# B&R Automation Studio project MotionTestBenchMaster (part 58)

```iecst
                               VAR_DOS_SEQ.Device.LSJ201.ALR := FALSE;                                                 (* STEP: 163 *)
                               VAR_DOS_SEQ.Device.LSJ201.WAIT_OFF := FALSE;
                               VAR_DOS_SEQ.Device.LSJ201.WAIT_ON := FALSE;

                               VAR_DOS_SEQ.Device.LSJ202.ALR := FALSE;                                                 (* STEP: 163 *)
                               VAR_DOS_SEQ.Device.LSJ202.WAIT_OFF := FALSE;
                               VAR_DOS_SEQ.Device.LSJ202.WAIT_ON := FALSE;

                               VAR_DOS_SEQ.Device.FSJ201.ALR := FALSE;                                                 (* STEP: 163 *)
                               VAR_DOS_SEQ.Device.FSJ201.WAIT_OFF := FALSE;
                               VAR_DOS_SEQ.Device.FSJ201.WAIT_ON := FALSE;

                               VAR_DOS_SEQ.Device.FSJ202.ALR := FALSE;                                                 (* STEP: 163 *)
                               VAR_DOS_SEQ.Device.FSJ202.WAIT_OFF := FALSE;
                               VAR_DOS_SEQ.Device.FSJ202.WAIT_ON := FALSE;

                               VAR_DOS_SEQ.Mem.PBAbortEnable := FALSE;                                                 (* STEP: 163 PB Abort Sequence Enable*)
                               VAR_DOS_SEQ.Mem.PBStopEnable := TRUE;                                                   (* STEP: 163 PB Stop Sequence Enable*)
                               VAR_DOS_SEQ.Mem.PBStartEnable := FALSE;                                                 (* STEP: 163 PB Start Sequence Enable*)
                               VAR_DOS_SEQ.Mem.ContainersStop := TRUE;                                                (* STEP: 163 *)
                               VAR_DOS_SEQ.Mem.MachineStart := FALSE;                                                  (* STEP: 163 *)
                               VAR_DOS_SEQ.Mem.MachineStop := FALSE;                                                   (* STEP: 163 *)
                               VAR_DOS_SEQ.Mem.DummyBottles := FALSE;                                                  (* STEP: 163 Dummy Bottle Install*)
                               VAR_DOS_SEQ.Mem.PositioningRequest := FALSE;                                            (* STEP: 163 Request of Cam Positioning at height SP of Sequncer*)
                               VAR_DOS_SEQ.Mem.COP_Cycle := FALSE;                                                     (* STEP: 163 COP Cycle Check Requested*)
                               VAR_DOS_SEQ.Mem.LapsCounter := FALSE;                                                   (* STEP: 163 *)
                               VAR_DOS_SEQ.Mem.ValveOpening := FALSE;                                                  (* STEP: 163 *)
                               VAR_DOS_SEQ.Mem.CopAfterCipRequest := FALSE;                                            (* STEP: 163 Request Of Cop After Cip*)

                               VAR_DOS_SEQ.ITC.CIP_CleaningRequest := FALSE;                                           (* STEP: 163 To CIP -> Request of Solution Sending*)
                               VAR_DOS_SEQ.ITC.CIP_Alarm := FALSE;                                                     (* STEP: 163 To CIP -> Critical Alarm Present*)
                               VAR_DOS_SEQ.ITC.CIP_RinseEnded := FALSE;                                                (* STEP: 163 To CIP -> Rinse Finished*)
                               VAR_DOS_SEQ.ITC.CIP_ChangeEnded := FALSE;                                               (* STEP: 163 To CIP -> Change Finished*)
                               VAR_DOS_SEQ.ITC.CIP_DrainRunning := FALSE;                                              (* STEP: 163 To CIP -> Drain Cycle Running*)
                               VAR_DOS_SEQ.ITC.CIP_RinseRunning := FALSE;                                              (* STEP: 163 To CIP -> Rinse Cycle Running*)
                               VAR_DOS_SEQ.ITC.CIP_CleaningRunning := FALSE;                                           (* STEP: 163 To CIP -> Cleaning Cycle Running*)
                               VAR_DOS_SEQ.ITC.CIP_DrainEnded := FALSE;                                                (* STEP: 163 To CIP -> Drain Finished*)
                               VAR_DOS_SEQ.ITC.CIP_FloodingEnded := FALSE;                                             (* STEP: 163 To CIP -> Flooding Finished*)
                               VAR_DOS_SEQ.ITC.CIP_FlipEnable := FALSE;                                                (* STEP: 163 *)
                               VAR_DOS_SEQ.ITC.CIP_CycleEnded := FALSE;                                                (* STEP: 163 *)

                               VAR_DOS_SEQ.ITC.PROD_ReadyForHeating := FALSE;                                          (* STEP: 163 To PASTO -> Filler Ready for Production (Heating)*)
                               VAR_DOS_SEQ.ITC.PROD_DoserInTemperature := FALSE;                                       (* STEP: 163 To PASTO -> Filler Temperature OK (After Heating)*)
                               VAR_DOS_SEQ.ITC.PROD_ProductRequest := FALSE;                                           (* STEP: 163 To PASTO -> Product Request*)
                               VAR_DOS_SEQ.ITC.PROD_DoserOnFillingMode := FALSE;                                       (* STEP: 163 To PASTO -> Product Consumend -Filling Valve Opening*)
                               VAR_DOS_SEQ.ITC.PROD_EndProductionCompleted := FALSE;                                   (* STEP: 163 To PASTO -> End Production Done*)
                               VAR_DOS_SEQ.ITC.PROD_ProductRecoveryEnd := FALSE;                                       (* STEP: 163 To PASTO -> Product Recovery End*)
                               VAR_DOS_SEQ.ITC.PROD_WaterRequestAfterProd := FALSE;                                    (* STEP: 163 To PASTO -> Water Request For Filler Rinse Afetr Production*)

                       164: (* MOTORIZATION - Operation Completed *)

                               VAR_DOS_SEQ.Device.PPJ201_PID.PID_Enable := FALSE;                                      (* STEP: 164 Doser Recovery Pump*)
                               VAR_DOS_SEQ.Device.PPJ201_PID.PID_Mode := FALSE;
                               VAR_DOS_SEQ.Device.PPJ201_PID.Auto_SP_Value := 0;
                               VAR_DOS_SEQ.Device.PPJ201_PID.FIX_Value := 0;

                               VAR_DOS_SEQ.Device.PPJ202_PID.PID_Enable := FALSE;                                      (* STEP: 164 Doser Recovery Pump*)
                               VAR_DOS_SEQ.Device.PPJ202_PID.PID_Mode := FALSE;
                               VAR_DOS_SEQ.Device.PPJ202_PID.Auto_SP_Value := 0;
                               VAR_DOS_SEQ.Device.PPJ202_PID.FIX_Value := 0;

                               VAR_DOS_SEQ.Device.PPJ203_PID.PID_Enable := FALSE;                                      (* STEP: 164 Diaphragm Pump for Recovery pulp*)
                               VAR_DOS_SEQ.Device.PPJ203_PID.PID_Mode := FALSE;
                               VAR_DOS_SEQ.Device.PPJ203_PID.Auto_SP_Value := 0;
                               VAR_DOS_SEQ.Device.PPJ203_PID.FIX_Value := 0;

                               VAR_DOS_SEQ.Device.MMJ201_PID.PID_Enable := FALSE;                                      (* STEP: 164 Shaker Motor*)
                               VAR_DOS_SEQ.Device.MMJ201_PID.PID_Mode := FALSE;
                               VAR_DOS_SEQ.Device.MMJ201_PID.Auto_SP_Value := 0;
                               VAR_DOS_SEQ.Device.MMJ201_PID.FIX_Value := 0;

                               VAR_DOS_SEQ.Device.RVJ201_PID.PID_Enable := FALSE;                                      (* STEP: 164 *)
                               VAR_DOS_SEQ.Device.RVJ201_PID.PID_Mode := FALSE;
                               VAR_DOS_SEQ.Device.RVJ201_PID.Auto_SP_Value := 0;
                               VAR_DOS_SEQ.Device.RVJ201_PID.FIX_Value := 0;

                               VAR_DOS_SEQ.Device.AVJ201.AutoCnd := FALSE;                                             (* STEP: 164 Inlet Valve*)
                               VAR_DOS_SEQ.Device.AVJ201.EnableCnd := FALSE;
                               VAR_DOS_SEQ.Device.AVJ210.AutoCnd := FALSE;                                             (* STEP: 164 Washing Duct Valve*)
                               VAR_DOS_SEQ.Device.AVJ210.EnableCnd := FALSE;
                               VAR_DOS_SEQ.Device.AVJ211.AutoCnd := FALSE;                                             (* STEP: 164 Sprayball Valve*)
                               VAR_DOS_SEQ.Device.AVJ211.EnableCnd := FALSE;
                               VAR_DOS_SEQ.Device.AVJ212.AutoCnd := FALSE;                                             (* STEP: 164 *)
                               VAR_DOS_SEQ.Device.AVJ212.EnableCnd := FALSE;
                               VAR_DOS_SEQ.Device.AVJ215.AutoCnd := FALSE;                                             (* STEP: 164 Atmospheric drain valve*)
                               VAR_DOS_SEQ.Device.AVJ215.EnableCnd := FALSE;
                               VAR_DOS_SEQ.Device.AVJ216.AutoCnd := FALSE;                                             (* STEP: 164 Recirculation Valve*)
                               VAR_DOS_SEQ.Device.AVJ216.EnableCnd := FALSE;
                               VAR_DOS_SEQ.Device.AVJ217.AutoCnd := FALSE;                                             (* STEP: 164 Tank Hema Drain Valve*)
                               VAR_DOS_SEQ.Device.AVJ217.EnableCnd := FALSE;
                               VAR_DOS_SEQ.Device.AVJ218.AutoCnd := FALSE;                                             (* STEP: 164 Recirculation Valve*)
                               VAR_DOS_SEQ.Device.AVJ218.EnableCnd := FALSE;
                               VAR_DOS_SEQ.Device.AVJ221.AutoCnd := FALSE;                                             (* STEP: 164 Inlet Loop Valve*)
                               VAR_DOS_SEQ.Device.AVJ221.EnableCnd := FALSE;
                               VAR_DOS_SEQ.Device.AVJ230.AutoCnd := FALSE;                                             (* STEP: 164 *)
                               VAR_DOS_SEQ.Device.AVJ230.EnableCnd := FALSE;
                               VAR_DOS_SEQ.Device.AVJ231.AutoCnd := FALSE;                                             (* STEP: 164 *)
                               VAR_DOS_SEQ.Device.AVJ231.EnableCnd := FALSE;
                               VAR_DOS_SEQ.Device.AVJ232.AutoCnd := FALSE;                                             (* STEP: 164 *)
                               VAR_DOS_SEQ.Device.AVJ232.EnableCnd := FALSE;
                               VAR_DOS_SEQ.Device.AVJ233.AutoCnd := FALSE;                                             (* STEP: 164 *)
                               VAR_DOS_SEQ.Device.AVJ233.EnableCnd := FALSE;
                               VAR_DOS_SEQ.Device.AVJ234.AutoCnd := FALSE;                                             (* STEP: 164 *)
                               VAR_DOS_SEQ.Device.AVJ234.EnableCnd := FALSE;
                               VAR_DOS_SEQ.Device.AVJ235.AutoCnd := FALSE;                                             (* STEP: 164 *)
                               VAR_DOS_SEQ.Device.AVJ235.EnableCnd := FALSE;

                               VAR_DOS_SEQ.Device.LTJ203.ALR_HighLimitEn := FALSE;                                     (* STEP: 164 Hema Tank Level*)
                               VAR_DOS_SEQ.Device.LTJ203.ALR_HighLimitSP := 0;
                               VAR_DOS_SEQ.Device.LTJ203.ALR_LowLimitEn := FALSE;
                               VAR_DOS_SEQ.Device.LTJ203.ALR_LowLimitSP := 0;
                               VAR_DOS_SEQ.Device.LTJ203.SP := 0;
                               VAR_DOS_SEQ.Device.LTJ203.CMP := 0;
                               VAR_DOS_SEQ.Device.LTJ203.MinDev := 0;
                               VAR_DOS_SEQ.Device.LTJ203.MaxDev := 0;

                               VAR_DOS_SEQ.Device.TTJ203.ALR_HighLimitEn := FALSE;                                     (* STEP: 164 Hema Tank Temperature*)
                               VAR_DOS_SEQ.Device.TTJ203.ALR_HighLimitSP := 0;
                               VAR_DOS_SEQ.Device.TTJ203.ALR_LowLimitEn := FALSE;
                               VAR_DOS_SEQ.Device.TTJ203.ALR_LowLimitSP := 0;
                               VAR_DOS_SEQ.Device.TTJ203.SP := 0;
                               VAR_DOS_SEQ.Device.TTJ203.CMP := 0;
                               VAR_DOS_SEQ.Device.TTJ203.MinDev := 0;
                               VAR_DOS_SEQ.Device.TTJ203.MaxDev := 0;

                               VAR_DOS_SEQ.Device.LSJ200.ALR := FALSE;                                                 (* STEP: 164 *)
                               VAR_DOS_SEQ.Device.LSJ200.WAIT_OFF := FALSE;
                               VAR_DOS_SEQ.Device.LSJ200.WAIT_ON := FALSE;

                               VAR_DOS_SEQ.Device.LSJ201.ALR := FALSE;                                                 (* STEP: 164 *)
                               VAR_DOS_SEQ.Device.LSJ201.WAIT_OFF := FALSE;
                               VAR_DOS_SEQ.Device.LSJ201.WAIT_ON := FALSE;

                               VAR_DOS_SEQ.Device.LSJ202.ALR := FALSE;                                                 (* STEP: 164 *)
                               VAR_DOS_SEQ.Device.LSJ202.WAIT_OFF := FALSE;
                               VAR_DOS_SEQ.Device.LSJ202.WAIT_ON := FALSE;

                               VAR_DOS_SEQ.Device.FSJ201.ALR := FALSE;                                                 (* STEP: 164 *)
                               VAR_DOS_SEQ.Device.FSJ201.WAIT_OFF := FALSE;
                               VAR_DOS_SEQ.Device.FSJ201.WAIT_ON := FALSE;

                               VAR_DOS_SEQ.Device.FSJ202.ALR := FALSE;                                                 (* STEP: 164 *)
                               VAR_DOS_SEQ.Device.FSJ202.WAIT_OFF := FALSE;
                               VAR_DOS_SEQ.Device.FSJ202.WAIT_ON := FALSE;

                               VAR_DOS_SEQ.Mem.PBAbortEnable := FALSE;                                                 (* STEP: 164 PB Abort Sequence Enable*)
                               VAR_DOS_SEQ.Mem.PBStopEnable := TRUE;                                                   (* STEP: 164 PB Stop Sequence Enable*)
                               VAR_DOS_SEQ.Mem.PBStartEnable := FALSE;                                                 (* STEP: 164 PB Start Sequence Enable*)
                               VAR_DOS_SEQ.Mem.ContainersStop := TRUE;                                                (* STEP: 164 *)
                               VAR_DOS_SEQ.Mem.MachineStart := FALSE;                                                  (* STEP: 164 *)
                               VAR_DOS_SEQ.Mem.MachineStop := FALSE;                                                   (* STEP: 164 *)
                               VAR_DOS_SEQ.Mem.DummyBottles := FALSE;                                                  (* STEP: 164 Dummy Bottle Install*)
                               VAR_DOS_SEQ.Mem.PositioningRequest := FALSE;                                            (* STEP: 164 Request of Cam Positioning at height SP of Sequncer*)
                               VAR_DOS_SEQ.Mem.COP_Cycle := FALSE;                                                     (* STEP: 164 COP Cycle Check Requested*)
                               VAR_DOS_SEQ.Mem.LapsCounter := FALSE;                                                   (* STEP: 164 *)
                               VAR_DOS_SEQ.Mem.ValveOpening := FALSE;                                                  (* STEP: 164 *)
                               VAR_DOS_SEQ.Mem.CopAfterCipRequest := FALSE;                                            (* STEP: 164 Request Of Cop After Cip*)

                               VAR_DOS_SEQ.ITC.CIP_CleaningRequest := FALSE;                                           (* STEP: 164 To CIP -> Request of Solution Sending*)
                               VAR_DOS_SEQ.ITC.CIP_Alarm := FALSE;                                                     (* STEP: 164 To CIP -> Critical Alarm Present*)
                               VAR_DOS_SEQ.ITC.CIP_RinseEnded := FALSE;                                                (* STEP: 164 To CIP -> Rinse Finished*)
                               VAR_DOS_SEQ.ITC.CIP_ChangeEnded := FALSE;                                               (* STEP: 164 To CIP -> Change Finished*)
                               VAR_DOS_SEQ.ITC.CIP_DrainRunning := FALSE;                                              (* STEP: 164 To CIP -> Drain Cycle Running*)
                               VAR_DOS_SEQ.ITC.CIP_RinseRunning := FALSE;                                              (* STEP: 164 To CIP -> Rinse Cycle Running*)
                               VAR_DOS_SEQ.ITC.CIP_CleaningRunning := FALSE;                                           (* STEP: 164 To CIP -> Cleaning Cycle Running*)
                               VAR_DOS_SEQ.ITC.CIP_DrainEnded := FALSE;                                                (* STEP: 164 To CIP -> Drain Finished*)
                               VAR_DOS_SEQ.ITC.CIP_FloodingEnded := FALSE;                                             (* STEP: 164 To CIP -> Flooding Finished*)
                               VAR_DOS_SEQ.ITC.CIP_FlipEnable := FALSE;                                                (* STEP: 164 *)
                               VAR_DOS_SEQ.ITC.CIP_CycleEnded := FALSE;                                                (* STEP: 164 *)

                               VAR_DOS_SEQ.ITC.PROD_ReadyForHeating := FALSE;                                          (* STEP: 164 To PASTO -> Filler Ready for Production (Heating)*)
                               VAR_DOS_SEQ.ITC.PROD_DoserInTemperature := FALSE;                                       (* STEP: 164 To PASTO -> Filler Temperature OK (After Heating)*)
                               VAR_DOS_SEQ.ITC.PROD_ProductRequest := FALSE;                                           (* STEP: 164 To PASTO -> Product Request*)
                               VAR_DOS_SEQ.ITC.PROD_DoserOnFillingMode := FALSE;                                       (* STEP: 164 To PASTO -> Product Consumend -Filling Valve Opening*)
                               VAR_DOS_SEQ.ITC.PROD_EndProductionCompleted := FALSE;                                   (* STEP: 164 To PASTO -> End Production Done*)
                               VAR_DOS_SEQ.ITC.PROD_ProductRecoveryEnd := FALSE;                                       (* STEP: 164 To PASTO -> Product Recovery End*)
                               VAR_DOS_SEQ.ITC.PROD_WaterRequestAfterProd := FALSE;                                    (* STEP: 164 To PASTO -> Water Request For Filler Rinse Afetr Production*)

                       165: (* MOTORIZATION - Error *)

                               VAR_DOS_SEQ.Device.PPJ201_PID.PID_Enable := FALSE;                                      (* STEP: 165 Doser Recovery Pump*)
                               VAR_DOS_SEQ.Device.PPJ201_PID.PID_Mode := FALSE;
                               VAR_DOS_SEQ.Device.PPJ201_PID.Auto_SP_Value := 0;
                               VAR_DOS_SEQ.Device.PPJ201_PID.FIX_Value := 0;

                               VAR_DOS_SEQ.Device.PPJ202_PID.PID_Enable := FALSE;                                      (* STEP: 165 Doser Recovery Pump*)
                               VAR_DOS_SEQ.Device.PPJ202_PID.PID_Mode := FALSE;
                               VAR_DOS_SEQ.Device.PPJ202_PID.Auto_SP_Value := 0;
                               VAR_DOS_SEQ.Device.PPJ202_PID.FIX_Value := 0;

                               VAR_DOS_SEQ.Device.PPJ203_PID.PID_Enable := FALSE;                                      (* STEP: 165 Diaphragm Pump for Recovery pulp*)
                               VAR_DOS_SEQ.Device.PPJ203_PID.PID_Mode := FALSE;
                               VAR_DOS_SEQ.Device.PPJ203_PID.Auto_SP_Value := 0;
                               VAR_DOS_SEQ.Device.PPJ203_PID.FIX_Value := 0;

                               VAR_DOS_SEQ.Device.MMJ201_PID.PID_Enable := FALSE;                                      (* STEP: 165 Shaker Motor*)
                               VAR_DOS_SEQ.Device.MMJ201_PID.PID_Mode := FALSE;
                               VAR_DOS_SEQ.Device.MMJ201_PID.Auto_SP_Value := 0;
                               VAR_DOS_SEQ.Device.MMJ201_PID.FIX_Value := 0;

                               VAR_DOS_SEQ.Device.RVJ201_PID.PID_Enable := FALSE;                                      (* STEP: 165 *)
                               VAR_DOS_SEQ.Device.RVJ201_PID.PID_Mode := FALSE;
                               VAR_DOS_SEQ.Device.RVJ201_PID.Auto_SP_Value := 0;
                               VAR_DOS_SEQ.Device.RVJ201_PID.FIX_Value := 0;

                               VAR_DOS_SEQ.Device.AVJ201.AutoCnd := FALSE;                                             (* STEP: 165 Inlet Valve*)
                               VAR_DOS_SEQ.Device.AVJ201.EnableCnd := FALSE;
                               VAR_DOS_SEQ.Device.AVJ210.AutoCnd := FALSE;                                             (* STEP: 165 Washing Duct Valve*)
                               VAR_DOS_SEQ.Device.AVJ210.EnableCnd := FALSE;
                               VAR_DOS_SEQ.Device.AVJ211.AutoCnd := FALSE;                                             (* STEP: 165 Sprayball Valve*)
                               VAR_DOS_SEQ.Device.AVJ211.EnableCnd := FALSE;
                               VAR_DOS_SEQ.Device.AVJ212.AutoCnd := FALSE;                                             (* STEP: 165 *)
                               VAR_DOS_SEQ.Device.AVJ212.EnableCnd := FALSE;
                               VAR_DOS_SEQ.Device.AVJ215.AutoCnd := FALSE;                                             (* STEP: 165 Atmospheric drain valve*)
                               VAR_DOS_SEQ.Device.AVJ215.EnableCnd := FALSE;
                               VAR_DOS_SEQ.Device.AVJ216.AutoCnd := FALSE;                                             (* STEP: 165 Recirculation Valve*)
                               VAR_DOS_SEQ.Device.AVJ216.EnableCnd := FALSE;
                               VAR_DOS_SEQ.Device.AVJ217.AutoCnd := FALSE;                                             (* STEP: 165 Tank Hema Drain Valve*)
                               VAR_DOS_SEQ.Device.AVJ217.EnableCnd := FALSE;
                               VAR_DOS_SEQ.Device.AVJ218.AutoCnd := FALSE;                                             (* STEP: 165 Recirculation Valve*)
                               VAR_DOS_SEQ.Device.AVJ218.EnableCnd := FALSE;
                               VAR_DOS_SEQ.Device.AVJ221.AutoCnd := FALSE;                                             (* STEP: 165 Inlet Loop Valve*)
                               VAR_DOS_SEQ.Device.AVJ221.EnableCnd := FALSE;
                               VAR_DOS_SEQ.Device.AVJ230.AutoCnd := FALSE;                                             (* STEP: 165 *)
                               VAR_DOS_SEQ.Device.AVJ230.EnableCnd := FALSE;
                               VAR_DOS_SEQ.Device.AVJ231.AutoCnd := FALSE;                                             (* STEP: 165 *)
                               VAR_DOS_SEQ.Device.AVJ231.EnableCnd := FALSE;
                               VAR_DOS_SEQ.Device.AVJ232.AutoCnd := FALSE;                                             (* STEP: 165 *)
                               VAR_DOS_SEQ.Device.AVJ232.EnableCnd := FALSE;
                               VAR_DOS_SEQ.Device.AVJ233.AutoCnd := FALSE;                                             (* STEP: 165 *)
                               VAR_DOS_SEQ.Device.AVJ233.EnableCnd := FALSE;
                               VAR_DOS_SEQ.Device.AVJ234.AutoCnd := FALSE;                                             (* STEP: 165 *)
                               VAR_DOS_SEQ.Device.AVJ234.EnableCnd := FALSE;
                               VAR_DOS_SEQ.Device.AVJ235.AutoCnd := FALSE;                                             (* STEP: 165 *)
                               VAR_DOS_SEQ.Device.AVJ235.EnableCnd := FALSE;

                               VAR_DOS_SEQ.Device.LTJ203.ALR_HighLimitEn := FALSE;                                     (* STEP: 165 Hema Tank Level*)
                               VAR_DOS_SEQ.Device.LTJ203.ALR_HighLimitSP := 0;
                               VAR_DOS_SEQ.Device.LTJ203.ALR_LowLimitEn := FALSE;
                               VAR_DOS_SEQ.Device.LTJ203.ALR_LowLimitSP := 0;
                               VAR_DOS_SEQ.Device.LTJ203.SP := 0;
                               VAR_DOS_SEQ.Device.LTJ203.CMP := 0;
                               VAR_DOS_SEQ.Device.LTJ203.MinDev := 0;
                               VAR_DOS_SEQ.Device.LTJ203.MaxDev := 0;

                               VAR_DOS_SEQ.Device.TTJ203.ALR_HighLimitEn := FALSE;                                     (* STEP: 165 Hema Tank Temperature*)
                               VAR_DOS_SEQ.Device.TTJ203.ALR_HighLimitSP := 0;
                               VAR_DOS_SEQ.Device.TTJ203.ALR_LowLimitEn := FALSE;
                               VAR_DOS_SEQ.Device.TTJ203.ALR_LowLimitSP := 0;
                               VAR_DOS_SEQ.Device.TTJ203.SP := 0;
                               VAR_DOS_SEQ.Device.TTJ203.CMP := 0;
                               VAR_DOS_SEQ.Device.TTJ203.MinDev := 0;
                               VAR_DOS_SEQ.Device.TTJ203.MaxDev := 0;

                               VAR_DOS_SEQ.Device.LSJ200.ALR := FALSE;                                                 (* STEP: 165 *)
                               VAR_DOS_SEQ.Device.LSJ200.WAIT_OFF := FALSE;
                               VAR_DOS_SEQ.Device.LSJ200.WAIT_ON := FALSE;

                               VAR_DOS_SEQ.Device.LSJ201.ALR := FALSE;                                                 (* STEP: 165 *)
                               VAR_DOS_SEQ.Device.LSJ201.WAIT_OFF := FALSE;
                               VAR_DOS_SEQ.Device.LSJ201.WAIT_ON := FALSE;

                               VAR_DOS_SEQ.Device.LSJ202.ALR := FALSE;                                                 (* STEP: 165 *)
                               VAR_DOS_SEQ.Device.LSJ202.WAIT_OFF := FALSE;
                               VAR_DOS_SEQ.Device.LSJ202.WAIT_ON := FALSE;

                               VAR_DOS_SEQ.Device.FSJ201.ALR := FALSE;                                                 (* STEP: 165 *)
                               VAR_DOS_SEQ.Device.FSJ201.WAIT_OFF := FALSE;
                               VAR_DOS_SEQ.Device.FSJ201.WAIT_ON := FALSE;

                               VAR_DOS_SEQ.Device.FSJ202.ALR := FALSE;                                                 (* STEP: 165 *)
                               VAR_DOS_SEQ.Device.FSJ202.WAIT_OFF := FALSE;
                               VAR_DOS_SEQ.Device.FSJ202.WAIT_ON := FALSE;

                               VAR_DOS_SEQ.Mem.PBAbortEnable := TRUE;                                                 (* STEP: 165 PB Abort Sequence Enable*)
                               VAR_DOS_SEQ.Mem.PBStopEnable := TRUE;                                                   (* STEP: 165 PB Stop Sequence Enable*)
                               VAR_DOS_SEQ.Mem.PBStartEnable := FALSE;                                                 (* STEP: 165 PB Start Sequence Enable*)
                               VAR_DOS_SEQ.Mem.ContainersStop := TRUE;                                                (* STEP: 165 *)
                               VAR_DOS_SEQ.Mem.MachineStart := FALSE;                                                  (* STEP: 165 *)
                               VAR_DOS_SEQ.Mem.MachineStop := FALSE;                                                   (* STEP: 165 *)
                               VAR_DOS_SEQ.Mem.DummyBottles := FALSE;                                                  (* STEP: 165 Dummy Bottle Install*)
                               VAR_DOS_SEQ.Mem.PositioningRequest := FALSE;                                            (* STEP: 165 Request of Cam Positioning at height SP of Sequncer*)
                               VAR_DOS_SEQ.Mem.COP_Cycle := FALSE;                                                     (* STEP: 165 COP Cycle Check Requested*)
                               VAR_DOS_SEQ.Mem.LapsCounter := FALSE;                                                   (* STEP: 165 *)
                               VAR_DOS_SEQ.Mem.ValveOpening := FALSE;                                                  (* STEP: 165 *)
                               VAR_DOS_SEQ.Mem.CopAfterCipRequest := FALSE;                                            (* STEP: 165 Request Of Cop After Cip*)

                               VAR_DOS_SEQ.ITC.CIP_CleaningRequest := FALSE;                                           (* STEP: 165 To CIP -> Request of Solution Sending*)
                               VAR_DOS_SEQ.ITC.CIP_Alarm := FALSE;                                                     (* STEP: 165 To CIP -> Critical Alarm Present*)
                               VAR_DOS_SEQ.ITC.CIP_RinseEnded := FALSE;                                                (* STEP: 165 To CIP -> Rinse Finished*)
                               VAR_DOS_SEQ.ITC.CIP_ChangeEnded := FALSE;                                               (* STEP: 165 To CIP -> Change Finished*)
                               VAR_DOS_SEQ.ITC.CIP_DrainRunning := FALSE;                                              (* STEP: 165 To CIP -> Drain Cycle Running*)
                               VAR_DOS_SEQ.ITC.CIP_RinseRunning := FALSE;                                              (* STEP: 165 To CIP -> Rinse Cycle Running*)
                               VAR_DOS_SEQ.ITC.CIP_CleaningRunning := FALSE;                                           (* STEP: 165 To CIP -> Cleaning Cycle Running*)
                               VAR_DOS_SEQ.ITC.CIP_DrainEnded := FALSE;                                                (* STEP: 165 To CIP -> Drain Finished*)
                               VAR_DOS_SEQ.ITC.CIP_FloodingEnded := FALSE;                                             (* STEP: 165 To CIP -> Flooding Finished*)
                               VAR_DOS_SEQ.ITC.CIP_FlipEnable := FALSE;                                                (* STEP: 165 *)
                               VAR_DOS_SEQ.ITC.CIP_CycleEnded := FALSE;                                                (* STEP: 165 *)

                               VAR_DOS_SEQ.ITC.PROD_ReadyForHeating := FALSE;                                          (* STEP: 165 To PASTO -> Filler Ready for Production (Heating)*)
                               VAR_DOS_SEQ.ITC.PROD_DoserInTemperature := FALSE;                                       (* STEP: 165 To PASTO -> Filler Temperature OK (After Heating)*)
                               VAR_DOS_SEQ.ITC.PROD_ProductRequest := FALSE;                                           (* STEP: 165 To PASTO -> Product Request*)
                               VAR_DOS_SEQ.ITC.PROD_DoserOnFillingMode := FALSE;                                       (* STEP: 165 To PASTO -> Product Consumend -Filling Valve Opening*)
                               VAR_DOS_SEQ.ITC.PROD_EndProductionCompleted := FALSE;                                   (* STEP: 165 To PASTO -> End Production Done*)
                               VAR_DOS_SEQ.ITC.PROD_ProductRecoveryEnd := FALSE;                                       (* STEP: 165 To PASTO -> Product Recovery End*)
                               VAR_DOS_SEQ.ITC.PROD_WaterRequestAfterProd := FALSE;                                    (* STEP: 165 To PASTO -> Water Request For Filler Rinse Afetr Production*)

                       166..169: (* Spare Steps *)

                       170: (* PRODUCTION - Doser Excluded *)

                               VAR_DOS_SEQ.Device.PPJ201_PID.PID_Enable := FALSE;                                      (* STEP: 170 Doser Recovery Pump*)
                               VAR_DOS_SEQ.Device.PPJ201_PID.PID_Mode := FALSE;
                               VAR_DOS_SEQ.Device.PPJ201_PID.Auto_SP_Value := 0;
                               VAR_DOS_SEQ.Device.PPJ201_PID.FIX_Value := 0;

                               VAR_DOS_SEQ.Device.PPJ202_PID.PID_Enable := FALSE;                                      (* STEP: 170 Doser Recovery Pump*)
                               VAR_DOS_SEQ.Device.PPJ202_PID.PID_Mode := FALSE;
                               VAR_DOS_SEQ.Device.PPJ202_PID.Auto_SP_Value := 0;
                               VAR_DOS_SEQ.Device.PPJ202_PID.FIX_Value := 0;

                               VAR_DOS_SEQ.Device.PPJ203_PID.PID_Enable := FALSE;                                      (* STEP: 170 Diaphragm Pump for Recovery pulp*)
                               VAR_DOS_SEQ.Device.PPJ203_PID.PID_Mode := FALSE;
                               VAR_DOS_SEQ.Device.PPJ203_PID.Auto_SP_Value := 0;
                               VAR_DOS_SEQ.Device.PPJ203_PID.FIX_Value := 0;

                               VAR_DOS_SEQ.Device.MMJ201_PID.PID_Enable := FALSE;                                      (* STEP: 170 Shaker Motor*)
                               VAR_DOS_SEQ.Device.MMJ201_PID.PID_Mode := FALSE;
                               VAR_DOS_SEQ.Device.MMJ201_PID.Auto_SP_Value := 0;
                               VAR_DOS_SEQ.Device.MMJ201_PID.FIX_Value := 0;

                               VAR_DOS_SEQ.Device.RVJ201_PID.PID_Enable := FALSE;                                      (* STEP: 170 *)
                               VAR_DOS_SEQ.Device.RVJ201_PID.PID_Mode := FALSE;
                               VAR_DOS_SEQ.Device.RVJ201_PID.Auto_SP_Value := 0;
                               VAR_DOS_SEQ.Device.RVJ201_PID.FIX_Value := 0;

                               VAR_DOS_SEQ.Device.AVJ201.AutoCnd := FALSE;                                             (* STEP: 170 Inlet Valve*)
                               VAR_DOS_SEQ.Device.AVJ201.EnableCnd := FALSE;
                               VAR_DOS_SEQ.Device.AVJ210.AutoCnd := FALSE;                                             (* STEP: 170 Washing Duct Valve*)
                               VAR_DOS_SEQ.Device.AVJ210.EnableCnd := FALSE;
                               VAR_DOS_SEQ.Device.AVJ211.AutoCnd := FALSE;                                             (* STEP: 170 Sprayball Valve*)
                               VAR_DOS_SEQ.Device.AVJ211.EnableCnd := FALSE;
                               VAR_DOS_SEQ.Device.AVJ212.AutoCnd := FALSE;                                             (* STEP: 170 *)
                               VAR_DOS_SEQ.Device.AVJ212.EnableCnd := FALSE;
                               VAR_DOS_SEQ.Device.AVJ215.AutoCnd := FALSE;                                             (* STEP: 170 Atmospheric drain valve*)
                               VAR_DOS_SEQ.Device.AVJ215.EnableCnd := FALSE;
                               VAR_DOS_SEQ.Device.AVJ216.AutoCnd := FALSE;                                             (* STEP: 170 Recirculation Valve*)
                               VAR_DOS_SEQ.Device.AVJ216.EnableCnd := FALSE;
                               VAR_DOS_SEQ.Device.AVJ217.AutoCnd := FALSE;                                             (* STEP: 170 Tank Hema Drain Valve*)
                               VAR_DOS_SEQ.Device.AVJ217.EnableCnd := FALSE;
                               VAR_DOS_SEQ.Device.AVJ218.AutoCnd := FALSE;                                             (* STEP: 170 Recirculation Valve*)
                               VAR_DOS_SEQ.Device.AVJ218.EnableCnd := FALSE;
                               VAR_DOS_SEQ.Device.AVJ221.AutoCnd := FALSE;                                             (* STEP: 170 Inlet Loop Valve*)
                               VAR_DOS_SEQ.Device.AVJ221.EnableCnd := FALSE;
                               VAR_DOS_SEQ.Device.AVJ230.AutoCnd := FALSE;                                             (* STEP: 170 *)
                               VAR_DOS_SEQ.Device.AVJ230.EnableCnd := FALSE;
                               VAR_DOS_SEQ.Device.AVJ231.AutoCnd := FALSE;                                             (* STEP: 170 *)
                               VAR_DOS_SEQ.Device.AVJ231.EnableCnd := FALSE;
                               VAR_DOS_SEQ.Device.AVJ232.AutoCnd := FALSE;                                             (* STEP: 170 *)
                               VAR_DOS_SEQ.Device.AVJ232.EnableCnd := FALSE;
                               VAR_DOS_SEQ.Device.AVJ233.AutoCnd := FALSE;                                             (* STEP: 170 *)
                               VAR_DOS_SEQ.Device.AVJ233.EnableCnd := FALSE;
                               VAR_DOS_SEQ.Device.AVJ234.AutoCnd := FALSE;                                             (* STEP: 170 *)
                               VAR_DOS_SEQ.Device.AVJ234.EnableCnd := FALSE;
                               VAR_DOS_SEQ.Device.AVJ235.AutoCnd := FALSE;                                             (* STEP: 170 *)
                               VAR_DOS_SEQ.Device.AVJ235.EnableCnd := FALSE;

                               VAR_DOS_SEQ.Device.LTJ203.ALR_HighLimitEn := FALSE;                                     (* STEP: 170 Hema Tank Level*)
                               VAR_DOS_SEQ.Device.LTJ203.ALR_HighLimitSP := 0;
                               VAR_DOS_SEQ.Device.LTJ203.ALR_LowLimitEn := FALSE;
                               VAR_DOS_SEQ.Device.LTJ203.ALR_LowLimitSP := 0;
                               VAR_DOS_SEQ.Device.LTJ203.SP := 0;
                               VAR_DOS_SEQ.Device.LTJ203.CMP := 0;
                               VAR_DOS_SEQ.Device.LTJ203.MinDev := 0;
                               VAR_DOS_SEQ.Device.LTJ203.MaxDev := 0;

                               VAR_DOS_SEQ.Device.TTJ203.ALR_HighLimitEn := FALSE;                                     (* STEP: 170 Hema Tank Temperature*)
                               VAR_DOS_SEQ.Device.TTJ203.ALR_HighLimitSP := 0;
                               VAR_DOS_SEQ.Device.TTJ203.ALR_LowLimitEn := FALSE;
                               VAR_DOS_SEQ.Device.TTJ203.ALR_LowLimitSP := 0;
                               VAR_DOS_SEQ.Device.TTJ203.SP := 0;
                               VAR_DOS_SEQ.Device.TTJ203.CMP := 0;
                               VAR_DOS_SEQ.Device.TTJ203.MinDev := 0;
                               VAR_DOS_SEQ.Device.TTJ203.MaxDev := 0;

                               VAR_DOS_SEQ.Device.LSJ200.ALR := FALSE;                                                 (* STEP: 170 *)
                               VAR_DOS_SEQ.Device.LSJ200.WAIT_OFF := FALSE;
                               VAR_DOS_SEQ.Device.LSJ200.WAIT_ON := FALSE;

                               VAR_DOS_SEQ.Device.LSJ201.ALR := FALSE;                                                 (* STEP: 170 *)
                               VAR_DOS_SEQ.Device.LSJ201.WAIT_OFF := FALSE;
                               VAR_DOS_SEQ.Device.LSJ201.WAIT_ON := FALSE;

                               VAR_DOS_SEQ.Device.LSJ202.ALR := FALSE;                                                 (* STEP: 170 *)
                               VAR_DOS_SEQ.Device.LSJ202.WAIT_OFF := FALSE;
                               VAR_DOS_SEQ.Device.LSJ202.WAIT_ON := FALSE;

                               VAR_DOS_SEQ.Device.FSJ201.ALR := FALSE;                                                 (* STEP: 170 *)
                               VAR_DOS_SEQ.Device.FSJ201.WAIT_OFF := FALSE;
                               VAR_DOS_SEQ.Device.FSJ201.WAIT_ON := FALSE;

                               VAR_DOS_SEQ.Device.FSJ202.ALR := FALSE;                                                 (* STEP: 170 *)
                               VAR_DOS_SEQ.Device.FSJ202.WAIT_OFF := FALSE;
                               VAR_DOS_SEQ.Device.FSJ202.WAIT_ON := FALSE;

                               VAR_DOS_SEQ.Mem.PBAbortEnable := FALSE;                                                 (* STEP: 170 PB Abort Sequence Enable*)
                               VAR_DOS_SEQ.Mem.PBStopEnable := FALSE;                                                   (* STEP: 170 PB Stop Sequence Enable*)
                               VAR_DOS_SEQ.Mem.PBStartEnable := FALSE;                                                 (* STEP: 170 PB Start Sequence Enable*)
                               VAR_DOS_SEQ.Mem.ContainersStop := FALSE;                                                (* STEP: 170 *)
                               VAR_DOS_SEQ.Mem.MachineStart := FALSE;                                                  (* STEP: 170 *)
                               VAR_DOS_SEQ.Mem.MachineStop := FALSE;                                                   (* STEP: 170 *)
                               VAR_DOS_SEQ.Mem.DummyBottles := FALSE;                                                  (* STEP: 170 Dummy Bottle Install*)
                               VAR_DOS_SEQ.Mem.PositioningRequest := FALSE;                                            (* STEP: 170 Request of Cam Positioning at height SP of Sequncer*)
                               VAR_DOS_SEQ.Mem.COP_Cycle := FALSE;                                                     (* STEP: 170 COP Cycle Check Requested*)
                               VAR_DOS_SEQ.Mem.LapsCounter := FALSE;                                                   (* STEP: 170 *)
                               VAR_DOS_SEQ.Mem.ValveOpening := FALSE;                                                  (* STEP: 170 *)
                               VAR_DOS_SEQ.Mem.CopAfterCipRequest := FALSE;                                            (* STEP: 170 Request Of Cop After Cip*)

                               VAR_DOS_SEQ.ITC.CIP_CleaningRequest := FALSE;                                           (* STEP: 170 To CIP -> Request of Solution Sending*)
                               VAR_DOS_SEQ.ITC.CIP_Alarm := FALSE;                                                     (* STEP: 170 To CIP -> Critical Alarm Present*)
                               VAR_DOS_SEQ.ITC.CIP_RinseEnded := FALSE;                                                (* STEP: 170 To CIP -> Rinse Finished*)
                               VAR_DOS_SEQ.ITC.CIP_ChangeEnded := FALSE;                                               (* STEP: 170 To CIP -> Change Finished*)
                               VAR_DOS_SEQ.ITC.CIP_DrainRunning := FALSE;                                              (* STEP: 170 To CIP -> Drain Cycle Running*)
                               VAR_DOS_SEQ.ITC.CIP_RinseRunning := FALSE;                                              (* STEP: 170 To CIP -> Rinse Cycle Running*)
                               VAR_DOS_SEQ.ITC.CIP_CleaningRunning := FALSE;                                           (* STEP: 170 To CIP -> Cleaning Cycle Running*)
                               VAR_DOS_SEQ.ITC.CIP_DrainEnded := FALSE;                                                (* STEP: 170 To CIP -> Drain Finished*)
                               VAR_DOS_SEQ.ITC.CIP_FloodingEnded := FALSE;                                             (* STEP: 170 To CIP -> Flooding Finished*)
                               VAR_DOS_SEQ.ITC.CIP_FlipEnable := FALSE;                                                (* STEP: 170 *)
                               VAR_DOS_SEQ.ITC.CIP_CycleEnded := FALSE;                                                (* STEP: 170 *)

                               VAR_DOS_SEQ.ITC.PROD_ReadyForHeating := FALSE;                                          (* STEP: 170 To PASTO -> Filler Ready for Production (Heating)*)
                               VAR_DOS_SEQ.ITC.PROD_DoserInTemperature := FALSE;                                       (* STEP: 170 To PASTO -> Filler Temperature OK (After Heating)*)
                               VAR_DOS_SEQ.ITC.PROD_ProductRequest := FALSE;                                           (* STEP: 170 To PASTO -> Product Request*)
                               VAR_DOS_SEQ.ITC.PROD_DoserOnFillingMode := FALSE;                                       (* STEP: 170 To PASTO -> Product Consumend -Filling Valve Opening*)
                               VAR_DOS_SEQ.ITC.PROD_EndProductionCompleted := FALSE;                                   (* STEP: 170 To PASTO -> End Production Done*)
                               VAR_DOS_SEQ.ITC.PROD_ProductRecoveryEnd := FALSE;                                       (* STEP: 170 To PASTO -> Product Recovery End*)
                               VAR_DOS_SEQ.ITC.PROD_WaterRequestAfterProd := FALSE;                                    (* STEP: 170 To PASTO -> Water Request For Filler Rinse Afetr Production*)

                       171..200: (* Spare Steps *)

               END_CASE
END_ACTION
```

#### DOS_StepStatus.st
```iecst
ACTION DOS_StepStatus:
	//MODE
	VAR_DOS_ModeWait					:= VAR_DOS_SeqPermanent.SeqActualStep = 0;
	VAR_DOS_ModeProduction				:= VAR_DOS_SeqPermanent.SeqMode1.0;
	VAR_DOS_ModeCip						:= VAR_DOS_SeqPermanent.SeqMode1.1;
	VAR_DOS_ModeRinse					:= VAR_DOS_SeqPermanent.SeqMode1.2;
	VAR_DOS_ModeDrain					:= VAR_DOS_SeqPermanent.SeqMode1.3;
	VAR_DOS_ModeCop						:= VAR_DOS_SeqPermanent.SeqMode1.4;
	VAR_DOS_ModePositioning				:= VAR_DOS_SeqPermanent.SeqMode1.5;
	VAR_DOS_ModeBypass					:= VAR_DOS_SeqPermanent.SeqMode1.6;
	VAR_DOS_ModePositionRequest			:= VAR_DOS_SeqPermanent.SeqMode1.7;
	VAR_DOS_ModeProductionExcluded		:= VAR_DOS_SeqPermanent.SeqMode1.8;
	VAR_DOS_MemProdDrain				:= VAR_DOS_SeqPermanent.SeqMode2.0;
	VAR_DOS_ModeWaitOperator			:= FALSE;

	VAR_DOS_MemDoserByPassed			:= VAR_DOS_SeqPermanent.SeqMode2.2;
	VAR_DOS_MemDoserIncluded			:= VAR_DOS_SeqPermanent.SeqMode2.3;

	VAR_DOS_MemDoserAxisOn				:= VAR_DOS_SeqPermanent.SeqMode2.4;
	VAR_DOS_MemDoserAxisOff				:= VAR_DOS_SeqPermanent.SeqMode2.5;
	VAR_DOS_MemFillerAxisOffReq			:= VAR_DOS_SeqPermanent.SeqMode2.6;

	//STEP PRODUCTION
	VAR_DOS_StepProdHeating				:= VAR_DOS_SEQ_Step.StepActual > 6 AND VAR_DOS_SeqActualStep < 15;
	VAR_DOS_StepProdProducing			:= VAR_DOS_SEQ_Step.StepActual = 35 OR VAR_DOS_SEQ_Step.StepActual = 37 OR VAR_DOS_SEQ_Step.StepActual = 38 OR
											VAR_DOS_SEQ_Step.StepActual = 22 OR VAR_DOS_SEQ_Step.StepActual = 23 OR VAR_DOS_SEQ_Step.StepActual = 30;
	VAR_DOS_StepProdLowLevel			:= VAR_DOS_SEQ_Step.StepActual = 37;
	VAR_DOS_StepProdRecovery			:= VAR_DOS_SEQ_Step.StepActual = 40;
	VAR_DOS_StepProdStopped				:= VAR_DOS_SEQ_Step.StepActual = 55;
	VAR_DOS_StepProdEndProduction		:= VAR_DOS_SEQ_Step.StepActual >= 46 AND VAR_DOS_SeqActualStep <= 52;
	VAR_DOS_StepProdAborted				:= VAR_DOS_SEQ_Step.StepActual = 0;

	//STEP CIP
	VAR_DOS_StepCipCleaning				:= VAR_DOS_SEQ_Step.StepActual > 73 AND VAR_DOS_SeqActualStep <=79;		//<	83
	VAR_DOS_StepCipDraining				:= VAR_DOS_SEQ_Step.StepActual >= 86 AND VAR_DOS_SeqActualStep <= 87;
	VAR_DOS_StepCipRecovery				:= VAR_DOS_SEQ_Step.StepActual = 82;
	VAR_DOS_StepCipStopped				:= VAR_DOS_SEQ_Step.StepActual = 95;
	VAR_DOS_StepCipAborted				:= VAR_DOS_SEQ_Step.StepActual = 96 OR VAR_DOS_SEQ_Step.StepActual = 0;
	VAR_DOS_StepCipEnded				:= VAR_DOS_SEQ_Step.StepActual = 88;
	VAR_DOS_StepCipFillerStartEnable	:= VAR_DOS_SEQ_Step.StepActual = 60 OR VAR_DOS_SeqActualStep = 61; //Segnale per SKID

	//STEP RINSE
	VAR_DOS_StepRinseReq				:=  VAR_DOS_SEQ_Step.StepActual >= 101 AND VAR_DOS_SeqActualStep <=106;
	VAR_DOS_StepRinseInExecution		:=  VAR_DOS_SEQ_Step.StepActual >= 101 AND VAR_DOS_SeqActualStep <=109;
	VAR_DOS_StepRinseAborted			:= VAR_DOS_SEQ_Step.StepActual = 0;
	VAR_DOS_StepRinseStopped			:= VAR_DOS_SEQ_Step.StepActual = 115;

	//STEP DRAIN
	VAR_DOS_StepDrainStopped			:= VAR_DOS_SEQ_Step.StepActual = 135;
	VAR_DOS_StepDrainAborted			:= VAR_DOS_SEQ_Step.StepActual = 0;

	//STEP COP
	VAR_DOS_StepCopRunning				:= VAR_DOS_SEQ_Step.StepActual = 90;

	//STEP BYPASS
	VAR_DOS_StepCamPositioning				:= VAR_DOS_SeqActualStep >= 150 AND VAR_DOS_SeqActualStep <= 155;
	VAR_DOS_StepCamPosRequest				:= VAR_DOS_SeqActualStep = 151;
	VAR_DOS_StepCamPosInProgress			:= VAR_DOS_SeqActualStep >= 151 AND VAR_DOS_SeqActualStep <= 154;
	VAR_DOS_StepBypassAborted				:= VAR_DOS_SeqActualStep = 0;

	//STEP MOTION
	VAR_DOS_StepMotorization				:= VAR_DOS_SeqActualStep >= 161 AND VAR_DOS_SeqActualStep <= 163;
END_ACTION
```

#### DOS_ValvesLogic.st
```iecst
ACTION DOS_ValvesLogic:

	VAR_DOS_ValveEnable := OPS.DataOut.EmergencyOk AND OPS.DataOut.GeneralAirOn AND OPS.DataOut.DoorsOk;

//AVJ201
	AVJ[201].IN_Enable		:= VAR_DOS_ValveEnable;
	AVJ[201].IN_AutoCnd		:= VAR_DOS_SEQ.Device.AVJ201.AutoCnd;
	AVJ[201].IN_EnableCnd	:= VAR_DOS_SEQ.Device.AVJ201.EnableCnd;
	AVJ[201].IN_Cnd 		:= (NOT LTJ[203].OUT_SpReached AND PstFlr.ProductAvailable AND VAR_DOS_StepProdProducing) OR
	                           (NOT LTJ[203].OUT_SpReached AND PstFlr.HeatingWithWater AND VAR_DOS_StepProdHeating) OR
                               (NOT LTJ[203].OUT_SpReached AND VAR_DOS_StepCipCleaning) OR
								(NOT LTJ[203].OUT_SpReached AND VAR_DOS_StepRinseReq) OR
								(NOT LTJ[203].OUT_SpReached AND VAR_DOS_SEQ_Step.StepActual = 46 AND  PstFlr.ProductAvailable); //46
	AVJ[201].IN_ManEn		:= TRUE;
	AVJ[201].IN_MaskEn		:= TRUE;

//AVJ210
	AVJ[210].IN_Enable		:= VAR_DOS_ValveEnable;
	AVJ[210].IN_AutoCnd		:= VAR_DOS_SEQ.Device.AVJ210.AutoCnd;
	AVJ[210].IN_EnableCnd	:= VAR_DOS_SEQ.Device.AVJ210.EnableCnd;
	AVJ[210].IN_Cnd 		:= FALSE;
	AVJ[210].IN_ManEn		:= TRUE;
	AVJ[210].IN_MaskEn		:= TRUE;

//AVJ211
	AVJ[211].IN_Enable		:= VAR_DOS_ValveEnable;
	AVJ[211].IN_AutoCnd		:= VAR_DOS_SEQ.Device.AVJ211.AutoCnd;
	AVJ[211].IN_EnableCnd	:= VAR_DOS_SEQ.Device.AVJ211.EnableCnd;
	AVJ[211].IN_Cnd 		:= NOT LTJ[203].OUT_HighLimit;
	AVJ[211].IN_ManEn		:= TRUE;
	AVJ[211].IN_MaskEn		:= TRUE;

//AVJ212
	AVJ[212].IN_Enable		:= VAR_DOS_ValveEnable;
	AVJ[212].IN_AutoCnd		:= VAR_DOS_SEQ.Device.AVJ212.AutoCnd;
	AVJ[212].IN_EnableCnd	:= VAR_DOS_SEQ.Device.AVJ212.EnableCnd;
	AVJ[212].IN_Cnd 		:= NOT LTJ[203].OUT_HighLimit;
	AVJ[212].IN_ManEn		:= TRUE;
	AVJ[212].IN_MaskEn		:= TRUE;

//AVJ215
	AVJ[215].IN_Enable		:= VAR_DOS_ValveEnable;
	AVJ[215].IN_AutoCnd		:= VAR_DOS_SEQ.Device.AVJ215.AutoCnd;
	AVJ[215].IN_EnableCnd	:= VAR_DOS_SEQ.Device.AVJ215.EnableCnd;
	AVJ[215].IN_Cnd 		:= FALSE;
	AVJ[215].IN_ManEn		:= TRUE;
	AVJ[215].IN_MaskEn		:= TRUE;

//AVJ216
	AVJ[216].IN_Enable		:= VAR_DOS_ValveEnable;
	AVJ[216].IN_AutoCnd		:= VAR_DOS_SEQ.Device.AVJ216.AutoCnd OR COP.DataOut.RcpActive ;
	AVJ[216].IN_EnableCnd	:= VAR_DOS_SEQ.Device.AVJ216.EnableCnd;
	AVJ[216].IN_Cnd 		:= FALSE;
	AVJ[216].IN_ManEn		:= TRUE;
	AVJ[216].IN_MaskEn		:= TRUE;

	//DYNAMIC COMMAND
	TMR_TON_FlipWait[0].IN	:= VAR_DOS_SEQ.Device.AVJ217.EnableCnd AND NOT TMR_TOF_FlipWork[0].Q;
	IF VAR_DOS_StepProdHeating THEN
		TMR_TON_FlipWait[0].PT	:= REAL_TO_TIME((HMI_PAM_3._614)*1000);
	ELSIF (VAR_DOS_StepCipCleaning OR VAR_DOS_StepRinseReq) THEN
		TMR_TON_FlipWait[0].PT	:= REAL_TO_TIME((HMI_PAM_3._637)*1000);
	END_IF
	TMR_TON_FlipWait[0]();

	TMR_TOF_FlipWork[0].IN := TMR_TON_FlipWait[0].Q;
	IF VAR_DOS_StepProdHeating THEN
		TMR_TOF_FlipWork[0].PT := REAL_TO_TIME((HMI_PAM_3._613)*1000); //[ms]*1000
	ELSIF (VAR_DOS_StepCipCleaning OR VAR_DOS_StepRinseReq) THEN
		TMR_TOF_FlipWork[0].PT := REAL_TO_TIME((HMI_PAM_3._636)*1000);
	END_IF
	TMR_TOF_FlipWork[0]();

	//AVJ217
	AVJ[217].IN_Enable		:= VAR_DOS_ValveEnable;
	AVJ[217].IN_AutoCnd		:= VAR_DOS_SEQ.Device.AVJ217.AutoCnd;
	AVJ[217].IN_EnableCnd	:= VAR_DOS_SEQ.Device.AVJ217.EnableCnd;
	AVJ[217].IN_Cnd 		:= TMR_TOF_FlipWork[0].Q;
	AVJ[217].IN_FlipEnable	:= FALSE;
	AVJ[217].IN_FlipRequest	:= FALSE;
	AVJ[217].IN_FlipTime	:= t#1s;
	AVJ[217].IN_ManEn		:= TRUE;
	AVJ[217].IN_MaskEn		:= TRUE;

//AVJ218
	AVJ[218].IN_Enable		:= VAR_DOS_ValveEnable;
	AVJ[218].IN_AutoCnd		:= VAR_DOS_SEQ.Device.AVJ218.AutoCnd;
	AVJ[218].IN_EnableCnd	:= VAR_DOS_SEQ.Device.AVJ218.EnableCnd;
	AVJ[218].IN_Cnd 		:= PPJ203.OUT_Cv > 0.2;
	AVJ[218].IN_ManEn		:= TRUE;
	AVJ[218].IN_MaskEn		:= TRUE;

//AVJ221
	AVJ[221].IN_Enable		:= TRUE;
	AVJ[221].IN_AutoCnd		:= NOT VAR_DOS_SEQ.Device.AVJ221.AutoCnd;	//NORMALLY OPEN - Sequencer managed as normally closed
	AVJ[221].IN_EnableCnd	:= VAR_DOS_SEQ.Device.AVJ221.EnableCnd;
	AVJ[221].IN_Cnd 		:= VAR_DOS_InletOpen OR AVJ[210].OUT_OpenedFiltered OR AVJ[211].OUT_OpenedFiltered;
	AVJ[221].IN_ManEn		:= TRUE;
	AVJ[221].IN_MaskEn		:= TRUE;

//AVJ230
	AVJ[230].IN_Enable		:= VAR_DOS_ValveEnable;
	AVJ[230].IN_AutoCnd		:= VAR_DOS_SEQ.Device.AVJ230.AutoCnd;
	AVJ[230].IN_EnableCnd	:= VAR_DOS_SEQ.Device.AVJ230.EnableCnd;
	AVJ[230].IN_Cnd 		:= NOT LSJ200H.OUT;
	AVJ[230].IN_ManEn		:= TRUE;
	AVJ[230].IN_MaskEn		:= TRUE;

//AVJ231
	AVJ[231].IN_Enable		:= VAR_DOS_ValveEnable;
	AVJ[231].IN_AutoCnd		:= VAR_DOS_SEQ.Device.AVJ231.AutoCnd;
	AVJ[231].IN_EnableCnd	:= VAR_DOS_SEQ.Device.AVJ231.EnableCnd;
	AVJ[231].IN_Cnd 		:= FALSE;
	AVJ[231].IN_ManEn		:= TRUE;
	AVJ[231].IN_MaskEn		:= TRUE;

//AVJ232
	AVJ[232].IN_Enable		:= VAR_DOS_ValveEnable;
	AVJ[232].IN_AutoCnd		:= VAR_DOS_SEQ.Device.AVJ232.AutoCnd OR COP.DataOut.RcpActive ;
	AVJ[232].IN_EnableCnd	:= VAR_DOS_SEQ.Device.AVJ232.EnableCnd;
	AVJ[232].IN_Cnd 		:= FALSE;
	AVJ[232].IN_ManEn		:= TRUE;
	AVJ[232].IN_MaskEn		:= TRUE;

//AVJ233
	AVJ[233].IN_Enable		:= VAR_DOS_ValveEnable;
	AVJ[233].IN_AutoCnd		:= VAR_DOS_SEQ.Device.AVJ233.AutoCnd OR PstFlr.CipReturnEnabled;
	AVJ[233].IN_EnableCnd	:= VAR_DOS_SEQ.Device.AVJ233.EnableCnd;
	AVJ[233].IN_Cnd 		:= FALSE;
	AVJ[233].IN_ManEn		:= TRUE;
	AVJ[233].IN_MaskEn		:= TRUE;

//AVJ234
	AVJ[234].IN_Enable		:= VAR_DOS_ValveEnable;
	AVJ[234].IN_AutoCnd		:= VAR_DOS_SEQ.Device.AVJ234.AutoCnd;
	AVJ[234].IN_EnableCnd	:= VAR_DOS_SEQ.Device.AVJ234.EnableCnd;
	AVJ[234].IN_Cnd 		:= FALSE;
	AVJ[234].IN_ManEn		:= TRUE;
	AVJ[234].IN_MaskEn		:= TRUE;

//AVJ235
	AVJ[235].IN_Enable		:= VAR_DOS_ValveEnable;
	AVJ[235].IN_AutoCnd		:= VAR_DOS_SEQ.Device.AVJ235.AutoCnd;
	AVJ[235].IN_EnableCnd	:= VAR_DOS_SEQ.Device.AVJ235.EnableCnd;
	AVJ[235].IN_Cnd 		:= FALSE;
	AVJ[235].IN_ManEn		:= TRUE;
	AVJ[235].IN_MaskEn		:= TRUE;

	//RVJ201
	RVJ[201].IN_Enable			:= VAR_DOS_ValveEnable;
	RVJ[201].IN_AutoCnd			:= RVJ[201].IN_Enable;
	//RVJ[201].IN_AutoVal 	:= FB_PID_RVJ201.OUT; //v1.0 : SEE TNK_ValvesFB.st
	RVJ[201].IN_MaskEn			:= RVJ[201].IN_ConfigPositionAnalogFBK;

	//PDO_YV65 FILIPPO TO DELETE
	PDO_YV65.IN_ConfigPresent := TRUE;
	PDO_YV65.IN_Enable		:= VAR_DOS_ValveEnable AND VAR_DOS_PumpEnable;
	PDO_YV65.IN_AutoCnd		:= PPJ203.IN_Enable AND VAR_DOS_SEQ.Device.PPJ203_PID.PID_Enable;
	PDO_YV65.IN_EnableCnd	:= FALSE;
	PDO_YV65.IN_Cnd 		:= FALSE;
	PDO_YV65.IN_ManEn		:= TRUE;
	PDO_YV65.IN_MaskEn		:= TRUE;

	//PDO_YV5 _211CPF
	_211CPF.IN_Enable		:= VAR_DOS_ValveEnable AND VAR_DOS_ModeCop;
	_211CPF.IN_EnableCnd	:= FALSE;
	_211CPF.IN_Cnd 			:= FALSE;
	_211CPF.IN_ManEn		:= FALSE;
	_211CPF.IN_MaskEn		:= FALSE;

END_ACTION
```

#### DOS_ModulatingPID.st
```iecst
ACTION DOS_ModulatingPID:
//RVJ201
	VAR_DOS_RVJ201Auto	:= NOT HMI_RVJ[201].ManOff AND NOT HMI_RVJ[201].ManOn;

	FB_PID_RVJ201[PID_MODE_PRD].IN_ConfigPresent	:= RVJ[201].IN_ConfigPresent;
	FB_PID_RVJ201[PID_MODE_PRD].IN_FixOut			:= RVJ[201].IN_Enable AND NOT VAR_DOS_SEQ.Device.RVJ201_PID.PID_Mode AND VAR_DOS_RVJ201Auto;
	FB_PID_RVJ201[PID_MODE_PRD].IN_Auto				:= RVJ[201].IN_Enable AND VAR_DOS_SEQ.Device.RVJ201_PID.PID_Mode AND VAR_DOS_RVJ201Auto;

	FB_PID_RVJ201[PID_MODE_PRD](
	IN_ConfigPresent	:= FB_PID_RVJ201[PID_MODE_PRD].IN_ConfigPresent,
	IN_Reverse 			:= TRUE,
	IN_Gain 			:= 2.0,//CREA PAM
	IN_TI 				:= 1.0,
	IN_TD 				:= 0.0,
	IN_PV 				:= LTJ[203].OUT_ActValue,
	IN_Auto				:= VAR_DOS_SEQ.Device.RVJ201_PID.PID_Enable AND FB_PID_RVJ201[PID_MODE_PRD].IN_Auto ,
	IN_FixOut			:= VAR_DOS_SEQ.Device.RVJ201_PID.PID_Enable AND FB_PID_RVJ201[PID_MODE_PRD].IN_FixOut,
	IN_FixOutValue 		:= VAR_DOS_SEQ.Device.RVJ201_PID.FIX_Value,
	IN_IntHold 			:= FALSE,
	IN_AutoSP 			:= VAR_DOS_SEQ.Device.RVJ201_PID.Auto_SP_Value,
	IN_Disv 			:= 0.0,
	IN_Slew 			:= FALSE,
	IN_SPSlew 			:= 0.0,
	IN_MaxScale			:= RVJ[201].IN_OutMax,
	IN_MinDev			:= 1.0,//PAM
	IN_MaxDev			:= 1.0,
	IN_OutMin 			:= RVJ[201].IN_OutMin,
	IN_OutMax 			:= RVJ[201].IN_OutMax,
	IN_CycleTime 		:= T#200ms,
	IN_TIInit 			:= FALSE,
	IN_TIInitValue 		:= 0.0,
	HMI 				:= HMI_PID_RVJ[201].Mode[PID_MODE_PRD]
	);
END_ACTION
```

#### DOS_ValvesFlip.st
```iecst
ACTION DOS_ValvesFlip:
	//CONFIGURATION FILIPPO
//	VAR_BTC_Flip_RTInfo(enable:=TRUE);
//	VAR_BTC_Flip_CycleTime :=UDINT_TO_REAL(VAR_BTC_Flip_RTInfo.cycle_time)/1000000; //TASK CYCLE TIME EXPRESS IN µsec . VAR_Cycle IS CONVERTED IN s

	//SET VALVE TO USE IN THE SEQUENCE
	VAR_DOS_FlipSeqValve[0].Config  	:= FALSE;
	VAR_DOS_FlipSeqValve[1].Config 		:= AVJ[217].IN_ConfigPresent;
	VAR_DOS_FlipSeqValve[2].Config 		:= FALSE;
	VAR_DOS_FlipSeqValve[3].Config 		:= FALSE;
	VAR_DOS_FlipSeqValve[4].Config 		:= FALSE;
	VAR_DOS_FlipSeqValve[5].Config 		:= FALSE;
	VAR_DOS_FlipSeqValve[6].Config 		:= FALSE;
	VAR_DOS_FlipSeqValve[7].Config 		:= FALSE;

	//SET VALVE EXECUTION DONE
	VAR_DOS_FlipSeqValve[0].Executed 	:= FALSE;
	VAR_DOS_FlipSeqValve[1].Executed 	:= AVJ[217].OUT_FlipDone;
	VAR_DOS_FlipSeqValve[2].Executed 	:= FALSE;
	VAR_DOS_FlipSeqValve[3].Executed 	:= FALSE;
	VAR_DOS_FlipSeqValve[4].Executed 	:= FALSE;
	VAR_DOS_FlipSeqValve[5].Executed 	:= FALSE;
	VAR_DOS_FlipSeqValve[6].Executed 	:= FALSE;
	VAR_DOS_FlipSeqValve[7].Executed 	:= FALSE;

	//SET DELAY BEFORE TO EXECUTE NEXT PHASE
	VAR_DOS_FlipSeqValve[0].TimeDelay_SP 	:= 240.0; //DELAY IN s TO NEXT SEQUENCE
	VAR_DOS_FlipSeqValve[1].TimeDelay_SP 	:= 2.0; //DELAY IN s TO NEXT SEQUENCE
	VAR_DOS_FlipSeqValve[2].TimeDelay_SP 	:= 2.0; //DELAY IN s TO NEXT SEQUENCE
	VAR_DOS_FlipSeqValve[3].TimeDelay_SP 	:= 2.0; //DELAY IN s TO NEXT SEQUENCE
	VAR_DOS_FlipSeqValve[4].TimeDelay_SP 	:= 2.0; //DELAY IN s TO NEXT SEQUENCE
	VAR_DOS_FlipSeqValve[5].TimeDelay_SP 	:= 2.0; //DELAY IN s TO NEXT SEQUENCE
	VAR_DOS_FlipSeqValve[6].TimeDelay_SP 	:= 2.0; //DELAY IN s TO NEXT SEQUENCE
	VAR_DOS_FlipSeqValve[7].TimeDelay_SP 	:= 2.0; //DELAY IN s TO NEXT SEQUENCE

	VAR_DOS_FlipSeqStart 	:= FALSE;
	VAR_DOS_FlipSeqEnable 	:= FALSE;
	VAR_DOS_FlipSeqEnd 		:= FALSE;
	VAR_DOS_FlipSeqReset	:= FALSE;

	//SCROLL MANAGEMENT
	IF VAR_DOS_FlipSeqStart AND NOT VAR_DOS_FlipSeqEnd THEN
		IF VAR_DOS_FlipSeqValve[VAR_DOS_FlipIndex].Config AND NOT VAR_DOS_FlipSeqValve[VAR_DOS_FlipIndex].SequenceDone THEN
			IF VAR_DOS_FlipSeqValve[VAR_DOS_FlipIndex].Done THEN	//OPENING EXECUTED
				VAR_DOS_FlipSeqValve[VAR_DOS_FlipIndex].TimeDelay_PV := VAR_DOS_FlipSeqValve[VAR_DOS_FlipIndex].TimeDelay_PV + VAR_DOS_Flip_CycleTime; 	//DELAY TIME COUNTING
			ELSE
				VAR_DOS_FlipSeqValve[VAR_DOS_FlipIndex].Request:= VAR_DOS_FlipSeqEnable AND NOT VAR_DOS_FlipSeqValve[VAR_DOS_FlipIndex].Executed; 		//REQUEST TO VALVE
				VAR_DOS_FlipSeqValve[VAR_DOS_FlipIndex].Done	:= VAR_DOS_FlipSeqValve[VAR_DOS_FlipIndex].Executed;			//EXECUTION REGISTERED
			END_IF

			IF VAR_DOS_FlipSeqValve[VAR_DOS_FlipIndex].TimeDelay_PV > VAR_DOS_FlipSeqValve[VAR_DOS_FlipIndex].TimeDelay_SP THEN	//DELAY PV > DELAY SP -> SEQUENCE DONE
				VAR_DOS_FlipSeqValve[VAR_DOS_FlipIndex].SequenceDone := TRUE;													//VALVE Seq DONE
				VAR_DOS_FlipIndex := MIN(VAR_DOS_FlipIndex+1,VAR_DOS_FlipSeqMax);
			END_IF
		ELSE
			VAR_DOS_FlipSeqValve[VAR_DOS_FlipIndex].SequenceDone := TRUE;		//SEQUENCE CLOSED
			VAR_DOS_FlipIndex := MIN(VAR_DOS_FlipIndex+1,VAR_DOS_FlipSeqMax);	//INDEX INCREASE
		END_IF
	END_IF
	//END OF ONE SEQUENCE
	IF EDGEPOS(VAR_DOS_FlipSeqValve[VAR_DOS_FlipSeqMax].SequenceDone) THEN
		VAR_DOS_FlipSequenceRepetition	:= VAR_DOS_FlipSequenceRepetition+1;
		VAR_DOS_FlipIndex				:= 0;
		memset(ADR(VAR_DOS_FlipSeqValve),0,SIZEOF(VAR_DOS_FlipSeqValve));
	END_IF
	//CLEAN ALL
	IF EDGEPOS(VAR_DOS_FlipSeqReset)THEN	//SCROLL RESET																									//STRUCTURE CLEAN
		memset(ADR(VAR_DOS_FlipSeqValve),0,SIZEOF(VAR_DOS_FlipSeqValve));
		VAR_DOS_FlipIndex				:= 0;
		VAR_DOS_FlipSequenceRepetition	:= 0;
	END_IF
END_ACTION
```

#### DOS_ValvesFB.st
```iecst
ACTION DOS_ValvesFB:

//AVJ201
	AVJ[201](
	IN_ConfigPresent 	:= AVJ[201].IN_ConfigPresent,
	IN_Enable 			:= AVJ[201].IN_Enable,
	IN_AutoCnd 			:= AVJ[201].IN_AutoCnd,
	IN_EnableCnd 		:= AVJ[201].IN_EnableCnd,
	IN_Cnd 				:= AVJ[201].IN_Cnd,
	IN_FlipEnable 		:= FALSE,
	IN_FlipRequest		:= FALSE,
	IN_FlipTime 		:= T#500ms,
	IN_Reset 			:= VAR_DOS_PBResetEp,
	IN_HMIAutoForce 	:= NOT HMI_SS2P[SS2P_HMI_DeviceEnable].ON,
	IN_ManEn 			:= AVJ[201].IN_ManEn,
	IN_MaskEn 			:= AVJ[201].IN_MaskEn,
	IO 					:= IO_AVJ[201],
	HMI 				:= HMI_AVJ[201]
	);

//AVJ210
	AVJ[210](
	IN_ConfigPresent 	:= AVJ[210].IN_ConfigPresent,
	IN_Enable 			:= AVJ[210].IN_Enable,
	IN_AutoCnd 			:= AVJ[210].IN_AutoCnd,
	IN_EnableCnd 		:= AVJ[210].IN_EnableCnd,
	IN_Cnd 				:= AVJ[210].IN_Cnd,
	IN_FlipEnable 		:= FALSE,
	IN_FlipRequest		:= FALSE,
	IN_FlipTime 		:= T#500ms,
	IN_Reset 			:= VAR_DOS_PBResetEp,
	IN_HMIAutoForce 	:= NOT HMI_SS2P[SS2P_HMI_DeviceEnable].ON,
	IN_ManEn 			:= AVJ[210].IN_ManEn,
	IN_MaskEn 			:= AVJ[210].IN_MaskEn,
	IO 					:= IO_AVJ[210],
	HMI 				:= HMI_AVJ[210]
	);

//AVJ211
	AVJ[211](
	IN_ConfigPresent 	:= AVJ[211].IN_ConfigPresent,
	IN_Enable 			:= AVJ[211].IN_Enable,
	IN_AutoCnd 			:= AVJ[211].IN_AutoCnd,
	IN_EnableCnd 		:= AVJ[211].IN_EnableCnd,
	IN_Cnd 				:= AVJ[211].IN_Cnd,
	IN_FlipEnable 		:= FALSE,
	IN_FlipRequest		:= FALSE,
	IN_FlipTime 		:= T#500ms,
	IN_Reset 			:= VAR_DOS_PBResetEp,
	IN_HMIAutoForce 	:= NOT HMI_SS2P[SS2P_HMI_DeviceEnable].ON,
	IN_ManEn 			:= AVJ[211].IN_ManEn,
	IN_MaskEn 			:= AVJ[211].IN_MaskEn,
	IO 					:= IO_AVJ[211],
	HMI 				:= HMI_AVJ[211]
	);

//AVJ212
	AVJ[212](
	IN_ConfigPresent 	:= AVJ[212].IN_ConfigPresent,
	IN_Enable 			:= AVJ[212].IN_Enable,
	IN_AutoCnd 			:= AVJ[212].IN_AutoCnd,
	IN_EnableCnd 		:= AVJ[212].IN_EnableCnd,
	IN_Cnd 				:= AVJ[212].IN_Cnd,
	IN_FlipEnable 		:= FALSE,
	IN_FlipRequest		:= FALSE,
	IN_FlipTime 		:= T#500ms,
	IN_Reset 			:= VAR_DOS_PBResetEp,
	IN_HMIAutoForce 	:= NOT HMI_SS2P[SS2P_HMI_DeviceEnable].ON,
	IN_ManEn 			:= AVJ[212].IN_ManEn,
	IN_MaskEn 			:= AVJ[212].IN_MaskEn,
	IO 					:= IO_AVJ[212],
	HMI 				:= HMI_AVJ[212]
	);

//AVJ215
	AVJ[215](
	IN_ConfigPresent 	:= AVJ[215].IN_ConfigPresent,
	IN_Enable 			:= AVJ[215].IN_Enable,
	IN_AutoCnd 			:= AVJ[215].IN_AutoCnd,
	IN_EnableCnd 		:= AVJ[215].IN_EnableCnd,
	IN_Cnd 				:= AVJ[215].IN_Cnd,
	IN_FlipEnable 		:= FALSE,
	IN_FlipRequest		:= FALSE,
	IN_FlipTime 		:= T#500ms,
	IN_Reset 			:= VAR_DOS_PBResetEp,
	IN_HMIAutoForce 	:= NOT HMI_SS2P[SS2P_HMI_DeviceEnable].ON,
	IN_ManEn 			:= AVJ[215].IN_ManEn,
	IN_MaskEn 			:= AVJ[215].IN_MaskEn,
	IO 					:= IO_AVJ[215],
	HMI 				:= HMI_AVJ[215]
	);

//AVJ216
	AVJ[216](
	IN_ConfigPresent 	:= AVJ[216].IN_ConfigPresent,
	IN_Enable 			:= AVJ[216].IN_Enable,
	IN_AutoCnd 			:= AVJ[216].IN_AutoCnd,
	IN_EnableCnd 		:= AVJ[216].IN_EnableCnd,
	IN_Cnd 				:= AVJ[216].IN_Cnd,
	IN_FlipEnable 		:= FALSE,
	IN_FlipRequest		:= FALSE,
	IN_FlipTime 		:= T#500ms,
	IN_Reset 			:= VAR_DOS_PBResetEp,
	IN_HMIAutoForce 	:= NOT HMI_SS2P[SS2P_HMI_DeviceEnable].ON,
	IN_ManEn 			:= AVJ[216].IN_ManEn,
	IN_MaskEn 			:= AVJ[216].IN_MaskEn,
	IO 					:= IO_AVJ[216],
	HMI 				:= HMI_AVJ[216]
	);

//AVJ217
	AVJ[217](
	IN_ConfigPresent 	:= AVJ[217].IN_ConfigPresent,
	IN_Enable 			:= AVJ[217].IN_Enable,
	IN_AutoCnd 			:= AVJ[217].IN_AutoCnd,
	IN_EnableCnd 		:= AVJ[217].IN_EnableCnd,
	IN_Cnd 				:= AVJ[217].IN_Cnd,
	IN_FlipEnable 		:= AVJ[217].IN_FlipEnable,
	IN_FlipRequest		:= AVJ[217].IN_FlipRequest,
	IN_FlipTime 		:= AVJ[217].IN_FlipTime,
	IN_Reset 			:= VAR_DOS_PBResetEp,
	IN_HMIAutoForce 	:= NOT HMI_SS2P[SS2P_HMI_DeviceEnable].ON,
	IN_ManEn 			:= AVJ[217].IN_ManEn,
	IN_MaskEn 			:= AVJ[217].IN_MaskEn,
	IO 					:= IO_AVJ[217],
	HMI 				:= HMI_AVJ[217]
	);

//AVJ218
	AVJ[218](
	IN_ConfigPresent 	:= AVJ[218].IN_ConfigPresent,
	IN_Enable 			:= AVJ[218].IN_Enable,
	IN_AutoCnd 			:= AVJ[218].IN_AutoCnd,
	IN_EnableCnd 		:= AVJ[218].IN_EnableCnd,
	IN_Cnd 				:= AVJ[218].IN_Cnd,
	IN_FlipEnable 		:= FALSE,
	IN_FlipRequest		:= FALSE,
	IN_FlipTime 		:= T#500ms,
	IN_Reset 			:= VAR_DOS_PBResetEp,
	IN_HMIAutoForce 	:= NOT HMI_SS2P[SS2P_HMI_DeviceEnable].ON,
	IN_ManEn 			:= AVJ[218].IN_ManEn,
	IN_MaskEn 			:= AVJ[218].IN_MaskEn,
	IO 					:= IO_AVJ[218],
	HMI 				:= HMI_AVJ[218]
	);

//AVJ221
	AVJ[221](
	IN_ConfigPresent 	:= AVJ[221].IN_ConfigPresent,
	IN_Enable 			:= AVJ[221].IN_Enable,
	IN_AutoCnd 			:= AVJ[221].IN_AutoCnd,
	IN_EnableCnd 		:= AVJ[221].IN_EnableCnd,
	IN_Cnd 				:= AVJ[221].IN_Cnd,
	IN_FlipEnable 		:= FALSE,
	IN_FlipRequest		:= FALSE,
	IN_FlipTime 		:= T#500ms,
	IN_Reset 			:= VAR_DOS_PBResetEp,
	IN_HMIAutoForce 	:= NOT HMI_SS2P[SS2P_HMI_DeviceEnable].ON,
	IN_ManEn 			:= AVJ[221].IN_ManEn,
	IN_MaskEn 			:= AVJ[221].IN_MaskEn,
	IO 					:= IO_AVJ[221],
	HMI 				:= HMI_AVJ[221]
	);

//AVJ230
	AVJ[230](
	IN_ConfigPresent 	:= AVJ[230].IN_ConfigPresent,
	IN_Enable 			:= AVJ[230].IN_Enable,
	IN_AutoCnd 			:= AVJ[230].IN_AutoCnd,
	IN_EnableCnd 		:= AVJ[230].IN_EnableCnd,
	IN_Cnd 				:= AVJ[230].IN_Cnd,
	IN_FlipEnable 		:= FALSE,
	IN_FlipRequest		:= FALSE,
	IN_FlipTime 		:= T#500ms,
	IN_Reset 			:= VAR_DOS_PBResetEp,
	IN_HMIAutoForce 	:= NOT HMI_SS2P[SS2P_HMI_DeviceEnable].ON,
	IN_ManEn 			:= AVJ[230].IN_ManEn,
	IN_MaskEn 			:= AVJ[230].IN_MaskEn,
	IO 					:= IO_AVJ[230],
	HMI 				:= HMI_AVJ[230]
	);

//AVJ231
	AVJ[231](
	IN_ConfigPresent 	:= AVJ[231].IN_ConfigPresent,
	IN_Enable 			:= AVJ[231].IN_Enable,
	IN_AutoCnd 			:= AVJ[231].IN_AutoCnd,
	IN_EnableCnd 		:= AVJ[231].IN_EnableCnd,
	IN_Cnd 				:= AVJ[231].IN_Cnd,
	IN_FlipEnable 		:= FALSE,
	IN_FlipRequest		:= FALSE,
	IN_FlipTime 		:= T#500ms,
	IN_Reset 			:= VAR_DOS_PBResetEp,
	IN_HMIAutoForce 	:= NOT HMI_SS2P[SS2P_HMI_DeviceEnable].ON,
	IN_ManEn 			:= AVJ[231].IN_ManEn,
	IN_MaskEn 			:= AVJ[231].IN_MaskEn,
	IO 					:= IO_AVJ[231],
	HMI 				:= HMI_AVJ[231]
	);

//AVJ232
	AVJ[232](
	IN_ConfigPresent 	:= AVJ[232].IN_ConfigPresent,
	IN_Enable 			:= AVJ[232].IN_Enable,
	IN_AutoCnd 			:= AVJ[232].IN_AutoCnd,
	IN_EnableCnd 		:= AVJ[232].IN_EnableCnd,
	IN_Cnd 				:= AVJ[232].IN_Cnd,
	IN_FlipEnable 		:= FALSE,
	IN_FlipRequest		:= FALSE,
	IN_FlipTime 		:= T#500ms,
	IN_Reset 			:= VAR_DOS_PBResetEp,
	IN_HMIAutoForce 	:= NOT HMI_SS2P[SS2P_HMI_DeviceEnable].ON,
	IN_ManEn 			:= AVJ[232].IN_ManEn,
	IN_MaskEn 			:= AVJ[232].IN_MaskEn,
	IO 					:= IO_AVJ[232],
	HMI 				:= HMI_AVJ[232]
	);

//AVJ233
	AVJ[233](
	IN_ConfigPresent 	:= AVJ[233].IN_ConfigPresent,
	IN_Enable 			:= AVJ[233].IN_Enable,
	IN_AutoCnd 			:= AVJ[233].IN_AutoCnd,
	IN_EnableCnd 		:= AVJ[233].IN_EnableCnd,
	IN_Cnd 				:= AVJ[233].IN_Cnd,
	IN_FlipEnable 		:= FALSE,
	IN_FlipRequest		:= FALSE,
	IN_FlipTime 		:= T#500ms,
	IN_Reset 			:= VAR_DOS_PBResetEp,
	IN_HMIAutoForce 	:= NOT HMI_SS2P[SS2P_HMI_DeviceEnable].ON,
	IN_ManEn 			:= AVJ[233].IN_ManEn,
	IN_MaskEn 			:= AVJ[233].IN_MaskEn,
	IO 					:= IO_AVJ[233],
	HMI 				:= HMI_AVJ[233]
	);

//AVJ234
	AVJ[234](
	IN_ConfigPresent 	:= AVJ[234].IN_ConfigPresent,
	IN_Enable 			:= AVJ[234].IN_Enable,
	IN_AutoCnd 			:= AVJ[234].IN_AutoCnd,
	IN_EnableCnd 		:= AVJ[234].IN_EnableCnd,
	IN_Cnd 				:= AVJ[234].IN_Cnd,
	IN_FlipEnable 		:= FALSE,
	IN_FlipRequest		:= FALSE,
	IN_FlipTime 		:= T#500ms,
	IN_Reset 			:= VAR_DOS_PBResetEp,
	IN_HMIAutoForce 	:= NOT HMI_SS2P[SS2P_HMI_DeviceEnable].ON,
	IN_ManEn 			:= AVJ[234].IN_ManEn,
	IN_MaskEn 			:= AVJ[234].IN_MaskEn,
	IO 					:= IO_AVJ[234],
	HMI 				:= HMI_AVJ[234]
	);

//AVJ235
	AVJ[235](
	IN_ConfigPresent 	:= AVJ[235].IN_ConfigPresent,
	IN_Enable 			:= AVJ[235].IN_Enable,
	IN_AutoCnd 			:= AVJ[235].IN_AutoCnd,
	IN_EnableCnd 		:= AVJ[235].IN_EnableCnd,
	IN_Cnd 				:= AVJ[235].IN_Cnd,
	IN_FlipEnable 		:= FALSE,
	IN_FlipRequest		:= FALSE,
	IN_FlipTime 		:= T#500ms,
	IN_Reset 			:= VAR_DOS_PBResetEp,
	IN_HMIAutoForce 	:= NOT HMI_SS2P[SS2P_HMI_DeviceEnable].ON,
	IN_ManEn 			:= AVJ[235].IN_ManEn,
	IN_MaskEn 			:= AVJ[235].IN_MaskEn,
	IO 					:= IO_AVJ[235],
	HMI 				:= HMI_AVJ[235]
	);

	//VALVES STATUS CONTROL
	VAR_DOS_InletOpen	:= AVJ[201].IN_ConfigPresent AND AVJ[201].OUT_OpenedFiltered;

	VAR_DOS_LoopOpen 	:= AVJ[221].OUT_ClosedFiltered AND AVJ[221].IN_ConfigPresent; //Normaly open

	VAR_DOS_ReturnOpen	:= AVJ[218].IN_ConfigPresent AND AVJ[218].OUT_OpenedFiltered;

	//VALVE FAULT
	VAR_DOS_AVJ_ValveFault	:= FALSE;

	FOR VAR_DOS_ForIndex := MIN_CFG_AVx TO MAX_CFG_AVx DO
		IF AVJ[VAR_DOS_ForIndex].IN_ConfigPresent AND AVJ[VAR_DOS_ForIndex].OUT_Alarm THEN
			VAR_DOS_AVJ_ValveFault	:= TRUE;
		END_IF
	END_FOR
	//INLET CLOSE DUE TO A FAULT
	TMR_TON_InletSafetyDelay.IN := VAR_DOS_AVJ_ValveFault;
	TMR_TON_InletSafetyDelay.PT := T#2s;
	TMR_TON_InletSafetyDelay();

//	VAR_DOS_ProductInletSafety		:= TMR_TON_InletSafetyDelay.IN;
//	VAR_DOS_ProductInletSafetyDelay	:= TMR_TON_InletSafetyDelay.Q AND AVB[223].OUT_ClosedFiltered;

//RVJ201
		RVJ[201].IN_AutoVal 			:= FB_PID_RVJ201[PID_MODE_PRD].OUT;

		RVJ[201](
		IN_ConfigPresent				:= RVJ[201].IN_ConfigPresent,
		IN_Enable 						:= RVJ[201].IN_Enable,
		IN_AutoCnd 						:= RVJ[201].IN_AutoCnd,
		IN_AutoVal 						:= RVJ[201].IN_AutoVal,
		IN_OpeningRampEn 				:= FALSE,
		IN_OpeningRampValue 			:= 0.0,
		IN_ClosingRampEn 				:= OPS.DataOut.EmergencyOk,
		IN_ClosingRampValue 			:= 10.0,
		IN_OutMin 						:= 0.0,
		IN_OutMax 						:= 100.0, //FAI PAM
		IN_HMIAutoForce 				:= NOT HMI_SS2P[SS2P_HMI_DeviceEnable].ON,
		IN_ManEn 						:= TRUE,
		IN_MaskEn 						:= RVJ[201].IN_MaskEn,
		IN_Reset 						:= VAR_DOS_PBResetEp,
		IO 								:= IO_RVJ[201],
		HMI 							:= HMI_RVJ[201]
	);

//PDO_YV65 FILIPPO
	PDO_YV65(
	IN_ConfigPresent 	:= PDO_YV65.IN_ConfigPresent,
	IN_Enable 			:= PDO_YV65.IN_Enable,
	IN_AutoCnd 			:= PDO_YV65.IN_AutoCnd,
	IN_EnableCnd 		:= PDO_YV65.IN_EnableCnd,
	IN_Cnd 				:= PDO_YV65.IN_Cnd,
	IN_FlipEnable 		:= FALSE,
	IN_FlipRequest		:= FALSE,
	IN_FlipTime 		:= T#500ms,
	IN_Reset 			:= VAR_DOS_PBResetEp,
	IN_HMIAutoForce 	:= NOT HMI_SS2P[SS2P_HMI_DeviceEnable].ON,
	IN_ManEn 			:= PDO_YV65.IN_ManEn,
	IN_MaskEn 			:= PDO_YV65.IN_MaskEn,
	IO 					:= IO_PDO_YV65,
	HMI 				:= HMI_PDO_YV65
	);

	//PDO_YV5 _211CPF
	_211CPF(
	IN_ConfigPresent 	:= _211CPF.IN_ConfigPresent,
	IN_Enable 			:= _211CPF.IN_Enable,
	IN_AutoCnd 			:= _211CPF.IN_AutoCnd,
	IN_EnableCnd 		:= _211CPF.IN_EnableCnd,
	IN_Cnd 				:= _211CPF.IN_Cnd,
	IN_FlipEnable 		:= FALSE,
	IN_FlipRequest		:= FALSE,
	IN_FlipTime 		:= T#500ms,
	IN_Reset 			:= VAR_DOS_PBResetEp,
	IN_HMIAutoForce 	:= NOT HMI_SS2P[SS2P_HMI_DeviceEnable].ON,
	IN_ManEn 			:= VAR_DOS_MMF205.SensorHighPos AND VAR_DOS_MMF206.SensorHighPos,
	IN_MaskEn 			:= _211CPF.IN_MaskEn,
	IO 					:= IO_211CPF,
	HMI 				:= HMI_211CPF
	);

	//Batteria 209PUF
	IO_209PUF_1.0 := IO_211CPF.DO_Closed;	//DO-02
	IO_209PUF_1.1 := IO_211CPF.DO_Opened;	//DO-01
	IO_209PUF_1.2 := FALSE;					//DO-04
	IO_209PUF_1.3 := FALSE;					//DO-03
	IO_209PUF_1.4 := IO_AVJ[210].DO_Opened;	//DO-06
	IO_209PUF_1.5 := IO_AVJ[201].DO_Opened; //DO-05
	IO_209PUF_1.6 := IO_AVJ[217].DO_Opened;	//DO-08
	IO_209PUF_1.7 := IO_AVJ[211].DO_Opened;	//DO-07

	IO_209PUF_2.0 := IO_AVJ[235].DO_Opened;	//DO-10
	IO_209PUF_2.1 := IO_AVJ[230].DO_Opened;	//DO-09
	IO_209PUF_2.2 := FALSE;					//DO-12
	IO_209PUF_2.3 := FALSE;					//DO-11
	IO_209PUF_2.4 := FALSE;					//DO-14
	IO_209PUF_2.5 := FALSE;					//DO-13
	IO_209PUF_2.6 := IO_AVJ[216].DO_Opened;	//DO-16
	IO_209PUF_2.7 := IO_AVJ[215].DO_Opened;	//DO-15

	IO_209PUF_3.0 := IO_AVJ[232].DO_Opened;	//DO-18
	IO_209PUF_3.1 := IO_AVJ[231].DO_Opened;	//DO-17
	IO_209PUF_3.2 := IO_AVJ[234].DO_Opened; //DO-20
	IO_209PUF_3.3 := IO_AVJ[233].DO_Opened;	//DO-19
	IO_209PUF_3.4 := FALSE;					//DO-22
	IO_209PUF_3.5 := FALSE;					//DO-21
	IO_209PUF_3.6 := FALSE;					//DO-24
	IO_209PUF_3.7 := FALSE;					//DO-23

END_ACTION
```

#### DOS_PumpsLogic.st
```iecst
ACTION DOS_PumpsLogic:

	VAR_DOS_PumpEnable := OPS.DataOut.EmergencyOk AND OPS.DataOut.EnablePump(*AND ARIA OK ???*);

	//PPJ201
	PPJ[201].IN_Enable 			:= VAR_DOS_PumpEnable;
	PPJ[201].IN_AutoCnd 		:= VAR_DOS_SEQ.Device.PPJ201_PID.PID_Enable;
	PPJ[201].IN_AutoSpeed 		:= 5.0;

	//PPJ202
	PPJ[202].IN_Enable 			:= VAR_DOS_PumpEnable;
	PPJ[202].IN_AutoCnd 		:= VAR_DOS_SEQ.Device.PPJ202_PID.PID_Enable OR PstFlr.CipReturnEnabled; //segnali di CIP recovery RMA FILIPPO
	PPJ[202].IN_AutoSpeed 		:= VAR_DOS_SEQ.Device.PPJ202_PID.FIX_Value;

	//DYNAMIC COMMAND
	TMR_TOF_FlipWork[1].IN := TMR_TON_FlipWait[1].Q;
	IF VAR_DOS_StepProdHeating THEN
		TMR_TOF_FlipWork[1].PT	:= REAL_TO_TIME((HMI_PAM_3._611)*1000); //[ms] * 1000
	ELSIF (VAR_DOS_StepCipCleaning OR VAR_DOS_StepRinseReq) THEN
		TMR_TOF_FlipWork[1].PT	:= REAL_TO_TIME((HMI_PAM_3._634)*1000);
	END_IF
	TMR_TOF_FlipWork[1]();

	TMR_TON_FlipWait[1].IN	:= (VAR_DOS_StepProdHeating OR VAR_DOS_StepCipCleaning OR VAR_DOS_StepRinseReq) AND NOT TMR_TOF_FlipWork[1].Q;
	IF VAR_DOS_StepProdHeating THEN
		TMR_TON_FlipWait[1].PT	:= REAL_TO_TIME((HMI_PAM_3._612)*1000);
	ELSIF (VAR_DOS_StepCipCleaning OR VAR_DOS_StepRinseReq) THEN
		TMR_TON_FlipWait[1].PT	:= REAL_TO_TIME((HMI_PAM_3._635)*1000);
	END_IF
	TMR_TON_FlipWait[1]();

	//PPJ203
	PPJ203.IN_Enable 			:= VAR_DOS_PumpEnable;
	PPJ203.IN_AutoCnd 			:= TMR_TOF_FlipWork[1].Q OR VAR_DOS_StepProdRecovery; //PNEUMATIC PUMP --> PRODUCT RECOVERY
	PPJ203.IN_AutoVal			:= 2.0;
END_ACTION
```

#### DOS_PumpsPID.st
```iecst
ACTION DOS_PumpsPID:
//PPJ202 MANAGEMENT IN CIP
	FB_PID_PPJ202[PID_MODE_CIP].IN_ConfigPresent	:= PPJ[202].IN_ConfigPresent;
	FB_PID_PPJ202[PID_MODE_CIP].IN_Auto				:= FB_PID_PPJ202[PID_MODE_CIP].IN_ConfigPresent AND VAR_DOS_SEQ.Device.PPJ202_PID.PID_Enable AND NOT PPJ[202].OUT_DriveFault;
	FB_PID_PPJ202[PID_MODE_CIP].IN_FixOut			:= FB_PID_PPJ202[PID_MODE_CIP].IN_Auto AND NOT VAR_DOS_SEQ.Device.PPJ202_PID.PID_Mode;
	FB_PID_PPJ202[PID_MODE_CIP].IN_Auto				:= FB_PID_PPJ202[PID_MODE_CIP].IN_Auto AND VAR_DOS_SEQ.Device.PPJ202_PID.PID_Mode;
	FB_PID_PPJ202[PID_MODE_CIP].IN_PV				:= LTJ[203].OUT_ActValue;

	FB_PID_PPJ202[PID_MODE_CIP](
	IN_ConfigPresent	:= FB_PID_PPJ202[PID_MODE_CIP].IN_ConfigPresent,
	IN_Reverse 			:= FALSE,
	IN_Gain 			:= HMI_PAM_D1._616,
	IN_TI 				:= HMI_PAM_D1._617,
	IN_TD 				:= HMI_PAM_D1._618,
	IN_PV 				:= FB_PID_PPJ202[PID_MODE_CIP].IN_PV,
	IN_Auto				:= FB_PID_PPJ202[PID_MODE_CIP].IN_Auto,
	IN_FixOut			:= FB_PID_PPJ202[PID_MODE_CIP].IN_FixOut,
	IN_FixOutValue 		:= VAR_DOS_SEQ.Device.PPJ202_PID.FIX_Value,
	IN_IntHold 			:= FALSE,
	IN_AutoSP 			:= VAR_DOS_SEQ.Device.PPJ202_PID.Auto_SP_Value,
	IN_Disv 			:= 0.0, // A RICETTA
	IN_Slew 			:= HMI_PAM_D1._613>0.0,
	IN_SPSlew 			:= HMI_PAM_D1._613,
	IN_MaxScale			:= PPJ[202].IN_ScaleMax,
	IN_MinDev			:= HMI_PAM_D1._611,
	IN_MaxDev			:= HMI_PAM_D1._612,
	IN_OutMin 			:= PPJ[202].IN_FrequencyMin,
	IN_OutMax 			:= PPJ[202].IN_FrequencyMax,
	IN_CycleTime 		:= T#200ms,
	IN_TIInit 			:= FALSE,
	IN_TIInitValue 		:= 0.0,
	HMI 				:= HMI_PID_PPJ[202].Mode[PID_MODE_CIP]
	);
END_ACTION
```

#### DOS_PumpsFB.st
```iecst
ACTION DOS_PumpsFB:

//PPJ201
	PPJ[201](
	IN_Simulation 		:= FALSE,
	IN_ConfigPresent 	:= PPJ[201].IN_ConfigPresent,
	IN_Enable 			:= PPJ[201].IN_Enable,
	IN_AutoCnd 			:= PPJ[201].IN_AutoCnd,
	IN_AutoSpeed 		:= PPJ[201].IN_AutoSpeed,
	IN_Reverse 			:= FALSE,
	IN_FrequencyMin 	:= 0.0,
	IN_FrequencyMax 	:= 100.0,
	IN_ManEn 			:= TRUE,
	IN_MaskEn 			:= TRUE,
	IN_Reset 			:= VAR_DOS_PBResetEp,
	IN_HMIAutoForce 	:= NOT HMI_SS2P[SS2P_HMI_DeviceEnable].ON,
	IN_QuickStopCmd		:= NOT IO_PPJ[201].DI_SafetyEnable,
	IN_JOGMode 			:= FALSE,
	IN_JOGCnd 			:= FALSE,
	IN_CoastingCmd 		:= NOT OPS.DataOut.EnablePump,
	IN_FBKDelay 		:= T#1000MS,
	IN_SafetyCtrlEn 	:= FALSE,
	IN_ScaleMax 		:= 100.0,
	HMI_Danfoss 		:= HMI_VFD_PPJ[201],
	HMI_Motor 			:= HMI_PPJ[201],
	IO_DanfossFC280			:= IO_VFD_PPJ[201],
	IO_MotorFC280			:= IO_PPJ[201]
	);

//PPJ202
	PPJ[202](
	IN_Simulation 		:= FALSE,
	IN_ConfigPresent 	:= PPJ[202].IN_ConfigPresent,
	IN_Enable 			:= PPJ[202].IN_Enable,
	IN_AutoCnd 			:= PPJ[202].IN_AutoCnd,
	IN_AutoSpeed 		:= PPJ[202].IN_AutoSpeed,
	IN_Reverse 			:= FALSE,
	IN_FrequencyMin 	:= 0.0,
	IN_FrequencyMax 	:= 60.0,
	IN_ManEn 			:= TRUE,
	IN_MaskEn 			:= TRUE,
	IN_Reset 			:= VAR_DOS_PBResetEp,
	IN_HMIAutoForce 	:= NOT HMI_SS2P[SS2P_HMI_DeviceEnable].ON,
	IN_QuickStopCmd		:= NOT IO_PPJ[202].DI_SafetyEnable,
	IN_JOGMode 			:= FALSE,
	IN_JOGCnd 			:= FALSE,
	IN_CoastingCmd 		:= NOT OPS.DataOut.EnablePump,
	IN_FBKDelay 		:= T#1000MS,
	IN_SafetyCtrlEn 	:= FALSE,
	IN_ScaleMax 		:= 100.0,
	HMI_Danfoss 		:= HMI_VFD_PPJ[202],
	HMI_Motor 			:= HMI_PPJ[202],
	IO_DanfossFC280 			:= IO_VFD_PPJ[202],
	IO_MotorFC280			:= IO_PPJ[202]
	);

//PPJ203
	PPJ203(
	IN_ConfigPresent 	:= PPJ203.IN_ConfigPresent,
	IN_Enable 			:= PPJ203.IN_Enable,
	IN_AutoCnd 			:= PPJ203.IN_AutoCnd,
	IN_AutoVal 			:= PPJ203.IN_AutoVal,
	IN_OpeningRampEn 	:= FALSE,
	IN_OpeningRampValue := 0.0,
	IN_ClosingRampEn 	:= OPS.DataOut.EmergencyOk AND OPS.DataOut.DoorsOk,
	IN_ClosingRampValue := 10.0,
	IN_OutMin 			:= HMI_PAM_A1._400,
	IN_OutMax 			:= HMI_PAM_A1._401,  //6 bar
	IN_ManEn 			:= NOT PPJ203.IN_HMIAutoForce,
	IN_MaskEn 			:= TRUE,
	IN_Reset 			:= VAR_DOS_PBResetEp,
	IN_HMIAutoForce 	:= NOT HMI_SS2P[SS2P_HMI_DeviceEnable].ON,
	HMI 				:= HMI_PPJ203,
	IO		 			:= IO_PPJ203
	);

	PPJ203_AuxScale( //SENTRONIC Conversion from EngValue to %
	x	:= PPJ203.OUT_Cv,
	x1	:= 0.0,
	y1	:= 6553.4,
	x2	:= 6, //bar
	y2	:= 32767.0,
	);

	IO_PPJ203.AO_Raw := REAL_TO_INT(PPJ203_AuxScale.y);
END_ACTION
```

#### DOS_MotorsLogic.st
```iecst
ACTION DOS_MotorsLogic:
	VAR_DOS_AlarmActive := ALR[939].Active OR ALR[940].Active OR ALR[941].Active OR ALR[942].Active ;
	VAR_DOS_MotorEnable := OPS.DataOut.EmergencyOk AND OPS.DataOut.EnableDrive AND NOT VAR_DOS_AlarmActive;

	//MMJ201
	MMJ[201].IN_Enable 		:= VAR_DOS_MotorEnable AND REAL_TO_BOOL(HMI_PAR_1._217);
	MMJ[201].IN_AutoCnd 	:= MMJ[201].IN_Enable AND VAR_DOS_SEQ.Device.MMJ201_PID.PID_Mode;
	MMJ[201].IN_AutoSpeed	:= HMI_PAR_1._218;
	MMJ[201].IN_ManEn	 	:= TRUE;
	MMJ[201].IN_MaskEn	 	:= TRUE;

	//MMF205  FILIPPO
	MMF[205].IN_Enable 		:= VAR_DOS_MotorEnable AND (VAR_DOS_SEQ.Mem.PositioningRequest OR HMI_DOS_SS2P[SS2P_DOS_SelLiftMan].ON OR HMI_DOS_LiftPosition.Value <> 0 OR HMI_DOS_SS2P[SS2P_DOS_ProbeAdjustment].ON) ;
	MMF[205].IN_ManEn	 	:= TRUE;
	MMF[205].IN_MaskEn	 	:= TRUE;

	//MMF206
	MMF[206].IN_Enable 		:= VAR_DOS_MotorEnable AND (VAR_DOS_SEQ.Mem.PositioningRequest OR HMI_DOS_SS2P[SS2P_DOS_SelLiftMan].ON OR HMI_DOS_LiftPosition.Value <> 0 OR HMI_DOS_SS2P[SS2P_DOS_ProbeAdjustment].ON);
	MMF[206].IN_ManEn	 	:= TRUE;
	MMF[206].IN_MaskEn	 	:= TRUE;
END_ACTION
```

#### DOS_MotorsFB.st
```iecst
ACTION DOS_MotorsFB:

	MMJ[201](
	IN_ConfigPresent 	:= MMJ[201].IN_ConfigPresent,
	IN_Enable			:= MMJ[201].IN_Enable,
	IN_AutoCnd			:= MMJ[201].IN_AutoCnd,
	IN_AutoSpeed		:= MMJ[201].IN_AutoSpeed,
	IN_FrequencyMin		:= 0.0,
	IN_FrequencyMax		:= 60.0,
	IN_Reset			:= VAR_DOS_PBResetEp,
	IN_HMIAutoForce		:= NOT HMI_SS2P[SS2P_HMI_DeviceEnable].ON,
	IN_QuickStopCmd		:= NOT MMJ[201].IN_Enable,
	IN_ManEn			:= MMJ[201].IN_ManEn,
	IN_MaskEn			:= MMJ[201].IN_MaskEn,
	IN_ScaleMax			:= 60.0,
	HMI_Danfoss			:= HMI_VFD_MMJ[201],
	HMI_Motor			:= HMI_MMJ[201],
	IO_DanfossFC280		:= IO_VFD_MMJ[201],
	IO_MotorFC280		:= IO_MMJ[201]
	);

	MMF[205](
	IN_ConfigPresent 	:= MMF[205].IN_ConfigPresent,
	IN_Enable			:= MMF[205].IN_Enable,
	IN_AutoCnd			:= MMF[205].IN_AutoCnd,
	IN_AutoSpeed		:= LIMIT(MMF[205].IN_FrequencyMin, MAX(ABS(VAR_DOS_MMF205.SpActual[mm] - VAR_DOS_MMF205.PosActual[mm])*5.0, 10.0),MMF[205].IN_FrequencyMax),
	IN_FrequencyMin		:= 0.0,
	IN_FrequencyMax		:= 60.0,
	IN_Reverse			:= MMF[205].IN_Reverse,
	IN_Reset			:= VAR_DOS_PBResetEp,
	IN_HMIAutoForce		:= NOT HMI_SS2P[SS2P_HMI_DeviceEnable].ON,
	IN_QuickStopCmd		:= NOT MMF[205].IN_Enable,
	IN_ManEn			:= MMF[205].IN_ManEn,
	IN_MaskEn			:= MMF[205].IN_MaskEn,
	IN_ScaleMax			:= 100.0,
	HMI_Danfoss			:= HMI_VFD_MMF[205],
	HMI_Motor			:= HMI_MMF[205],
	IO_DanfossFC280		:= IO_VFD_MMF[205],
	IO_MotorFC280		:= IO_MMF[205]
	);

	MMF[206](
	IN_ConfigPresent 	:= MMF[206].IN_ConfigPresent,
	IN_Enable			:= MMF[206].IN_Enable,
	IN_AutoCnd			:= MMF[206].IN_AutoCnd,
	IN_AutoSpeed		:= LIMIT(MMF[206].IN_FrequencyMin, MAX(ABS(VAR_DOS_MMF206.SpActual[mm] - VAR_DOS_MMF206.PosActual[mm])*5.0, 10.0),MMF[206].IN_FrequencyMax),
	IN_FrequencyMin		:= 0.0,
	IN_FrequencyMax		:= 60.0,
	IN_Reverse			:= MMF[206].IN_Reverse,
	IN_Reset			:= VAR_DOS_PBResetEp,
	IN_HMIAutoForce		:= NOT HMI_SS2P[SS2P_HMI_DeviceEnable].ON,
	IN_QuickStopCmd		:= NOT MMF[206].IN_Enable,
	IN_ManEn			:= MMF[206].IN_ManEn,
	IN_MaskEn			:= MMF[206].IN_MaskEn,
	IN_ScaleMax			:= 100.0,
	HMI_Danfoss			:= HMI_VFD_MMF[206],
	HMI_Motor			:= HMI_MMF[206],
	IO_DanfossFC280			:= IO_VFD_MMF[206],
	IO_MotorFC280			:= IO_MMF[206]
	);

	VAR_DOS_MotorReady := VAR_DOS_MotorEnable AND NOT MMJ[201].OUT_DriveFault;
	VAR_DOS_MotorFault := VAR_DOS_MotorEnable AND MMJ[201].OUT_DriveFault;
END_ACTION
```
